KUKA KRL program: MyProgram_331().src

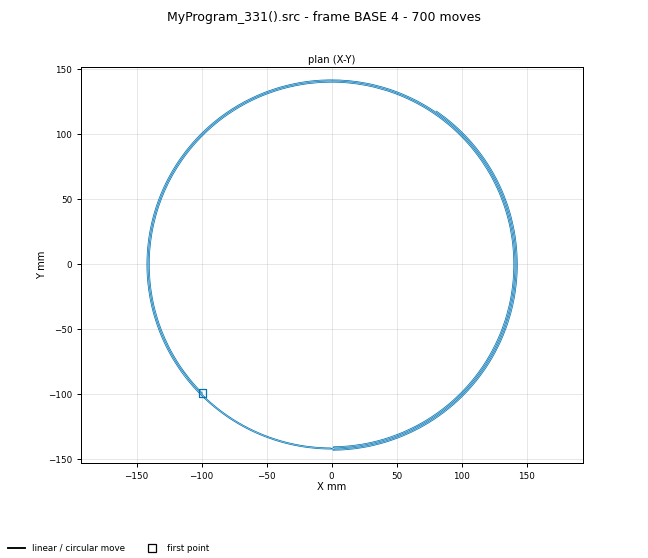
[picture p0: tool path of MyProgram_331().src in frame BASE 4, 700 of 700 moves have a stored position in this frame; points joined in program order, loops and branches not executed]
&ACCESS RVP
&REL 1
&PARAM TEMPLATE = C:\KRC\Roboter\Template\vorgabe
&PARAM EDITMASK = *
DEF MyProgram_331()
; ---- Setting reference (Base) ----
$BASE = BASE_DATA[4]

; --------------------------
; ---- Setting tool (TCP) ----
$TOOL = TOOL_DATA[3]
; --------------------------

$VEL.CP = VEL_APROX_PRINT
Startdeposition()
$VEL.CP = VEL_PRINT
LIN {X -99.2098,Y -99.0749,Z 188,A -128.7524,B 2.1644,C 0.244,E1 2.0676,E2 222.0446} C_DIS
LIN {X -102.5229,Y -95.6418,Z 188,A -131.099,B 2.1647,C 0.2414,E1 2.0629,E2 224.4451} C_DIS
LIN {X -106.6822,Y -90.9794,Z 188,A -133.6098,B 2.1653,C 0.2362,E1 2.0583,E2 226.9498} C_DIS
LIN {X -109.1006,Y -88.0645,Z 188,A -136.4618,B 2.1653,C 0.2366,E1 2.053,E2 229.9773} C_DIS
LIN {X -113.8783,Y -81.7931,Z 188,A -138.6384,B 2.1663,C 0.2268,E1 2.0496,E2 232.0127} C_DIS
LIN {X -116.0061,Y -78.7458,Z 188,A -140.3809,B 2.1666,C 0.224,E1 2.0468,E2 233.7852} C_DIS
LIN {X -118.4766,Y -74.9774,Z 188,A -142.4245,B 2.167,C 0.2203,E1 2.0437,E2 235.8555} C_DIS
LIN {X -121.0762,Y -70.7034,Z 188,A -144.5197,B 2.1674,C 0.2157,E1 2.0407,E2 237.9569} C_DIS
LIN {X -123.3353,Y -66.6846,Z 188,A -146.5209,B 2.1678,C 0.2114,E1 2.0379,E2 239.9733} C_DIS
LIN {X -125.1275,Y -63.2533,Z 188,A -148.0771,B 2.1682,C 0.2075,E1 2.036,E2 241.5254} C_DIS
LIN {X -126.6886,Y -60.0657,Z 188,A -149.6056,B 2.1685,C 0.2041,E1 2.0341,E2 243.0639} C_DIS
LIN {X -128.024,Y -57.1629,Z 188,A -151.3173,B 2.1688,C 0.2017,E1 2.0321,E2 244.8292} C_DIS
LIN {X -129.3709,Y -54.0455,Z 188,A -152.1682,B 2.1692,C 0.197,E1 2.0312,E2 245.6079} C_DIS
LIN {X -130.6105,Y -50.9774,Z 188,A -154.4978,B 2.1693,C 0.1957,E1 2.0287,E2 248.0671} C_DIS
LIN {X -132.2881,Y -46.4535,Z 188,A -155.8911,B 2.1699,C 0.1893,E1 2.0275,E2 249.3829} C_DIS
LIN {X -133.6605,Y -42.3408,Z 188,A -157.9257,B 2.1702,C 0.1852,E1 2.0257,E2 251.4516} C_DIS
LIN {X -134.6483,Y -39.0861,Z 188,A -159.3479,B 2.1705,C 0.1816,E1 2.0245,E2 252.8775} C_DIS
LIN {X -135.5192,Y -35.9493,Z 188,A -160.794,B 2.1708,C 0.1782,E1 2.0234,E2 254.3382} C_DIS
LIN {X -136.3712,Y -32.5697,Z 188,A -162.3237,B 2.1711,C 0.1746,E1 2.0224,E2 255.8812} C_DIS
LIN {X -137.2746,Y -28.5275,Z 188,A -164.3373,B 2.1714,C 0.1706,E1 2.0212,E2 257.9363} C_DIS
LIN {X -138.006,Y -24.7422,Z 188,A -165.7936,B 2.1718,C 0.166,E1 2.0205,E2 259.376} C_DIS
LIN {X -138.9297,Y -18.8902,Z 188,A -168.3319,B 2.1723,C 0.1595,E1 2.0194,E2 261.9286} C_DIS
LIN {X -139.6258,Y -12.7635,Z 188,A -171.0785,B 2.1727,C 0.1529,E1 2.0186,E2 264.7035} C_DIS
LIN {X -140.1378,Y -4.4233,Z 188,A -174.7771,B 2.1734,C 0.1439,E1 2.018,E2 268.4372} C_DIS
LIN {X -140.1787,Y 2.8448,Z 188,A -177.7366,B 2.1739,C 0.1356,E1 2.018,E2 271.3936} C_DIS
LIN {X -140.0302,Y 7.0299,Z 188,A -179.9971,B 2.1741,C 0.1317,E1 2.0182,E2 273.7241} C_DIS
LIN {X -139.782,Y 10.9262,Z 188,A 177.5471,B 2.1743,C 0.1288,E1 2.0189,E2 276.289} C_DIS
LIN {X -139.0996,Y 17.5935,Z 188,A 175.6823,B 2.1748,C 0.1196,E1 2.0194,E2 278.0404} C_DIS
LIN {X -138.1989,Y 23.6481,Z 188,A 172.9731,B 2.1752,C 0.1131,E1 2.0206,E2 280.7748} C_DIS
LIN {X -137.7195,Y 26.2897,Z 188,A 171.6814,B 2.1753,C 0.1104,E1 2.0212,E2 282.0906} C_DIS
LIN {X -136.8646,Y 30.4385,Z 188,A 169.7202,B 2.1755,C 0.106,E1 2.0224,E2 284.0801} C_DIS
LIN {X -135.2027,Y 37.1276,Z 188,A 166.9626,B 2.1759,C 0.0983,E1 2.0243,E2 286.8282} C_DIS
LIN {X -133.9173,Y 41.5233,Z 188,A 164.9103,B 2.1761,C 0.0936,E1 2.0259,E2 288.9021} C_DIS
LIN {X -132.743,Y 45.1415,Z 188,A 162.9991,B 2.1763,C 0.0902,E1 2.0277,E2 290.8574} C_DIS
LIN {X -131.3372,Y 49.0744,Z 188,A 161.3898,B 2.1764,C 0.0855,E1 2.0292,E2 292.4532} C_DIS
LIN {X -129.9982,Y 52.5188,Z 188,A 159.1417,B 2.1765,C 0.083,E1 2.0317,E2 294.7928} C_DIS
LIN {X -127.9992,Y 57.2184,Z 188,A 157.617,B 2.1768,C 0.0766,E1 2.0333,E2 296.2456} C_DIS
LIN {X -125.6046,Y 62.3001,Z 188,A 155.1346,B 2.177,C 0.0712,E1 2.0363,E2 298.7499} C_DIS
LIN {X -123.9945,Y 65.4459,Z 188,A 153.591,B 2.177,C 0.0679,E1 2.0383,E2 300.3049} C_DIS
LIN {X -121.9107,Y 69.2542,Z 188,A 150.9394,B 2.1771,C 0.0654,E1 2.0421,E2 303.0643} C_DIS
LIN {X -118.9504,Y 74.2235,Z 188,A 149.5886,B 2.1774,C 0.0578,E1 2.0439,E2 304.2876} C_DIS
LIN {X -114.8375,Y 80.4415,Z 188,A 145.4813,B 2.1774,C 0.0532,E1 2.0505,E2 308.5245} C_DIS
LIN {X -112.2475,Y 84.0171,Z 188,A 143.9413,B 2.1776,C 0.0486,E1 2.053,E2 310.0306} C_DIS
LIN {X -109.3338,Y 87.7754,Z 188,A 141.9211,B 2.1776,C 0.0446,E1 2.0565,E2 312.0589} C_DIS
LIN {X -106.409,Y 91.2989,Z 188,A 139.9971,B 2.1777,C 0.0409,E1 2.06,E2 313.9881} C_DIS
LIN {X -103.4782,Y 94.6081,Z 188,A 138.0511,B 2.1777,C 0.0376,E1 2.0636,E2 315.95} C_DIS
LIN {X -100.2471,Y 98.0248,Z 188,A 136.0546,B 2.1779,C 0.0341,E1 2.0675,E2 317.9543} C_DIS
LIN {X -96.8927,Y 101.3415,Z 188,A 134.0732,B 2.1779,C 0.0307,E1 2.0715,E2 319.9409} C_DIS
LIN {X -93.6314,Y 104.3622,Z 188,A 132.1553,B 2.1779,C 0.0277,E1 2.0755,E2 321.87} C_DIS
LIN {X -90.065,Y 107.455,Z 188,A 130.1679,B 2.1779,C 0.0245,E1 2.0797,E2 323.8631} C_DIS
LIN {X -86.4591,Y 110.3773,Z 188,A 128.1907,B 2.178,C 0.0217,E1 2.0841,E2 325.8488} C_DIS
LIN {X -82.9387,Y 113.0463,Z 188,A 126.1798,B 2.178,C 0.0195,E1 2.0886,E2 327.8835} C_DIS
LIN {X -78.3392,Y 116.2814,Z 188,A 124.065,B 2.178,C 0.0155,E1 2.0934,E2 329.9745} C_DIS
LIN {X -75.1994,Y 118.3365,Z 188,A 122.1429,B 2.178,C 0.0146,E1 2.0981,E2 331.9429} C_DIS
LIN {X -72.4256,Y 120.0535,Z 188,A 121.0215,B 2.178,C 0.0122,E1 2.1007,E2 333.0377} C_DIS
LIN {X -67.9868,Y 122.6217,Z 188,A 118.9997,B 2.178,C 0.0093,E1 2.1056,E2 335.0491} C_DIS
LIN {X -65.0011,Y 124.2281,Z 188,A 117.4444,B 2.1781,C 0.0083,E1 2.1095,E2 336.6242} C_DIS
LIN {X -60.611,Y 126.4281,Z 188,A 115.4931,B 2.1781,C 0.0059,E1 2.1144,E2 338.5675} C_DIS
LIN {X -56.8006,Y 128.1861,Z 188,A 113.2517,B 2.1781,C 0.0061,E1 2.1202,E2 340.8715} C_DIS
LIN {X -53.0986,Y 129.7645,Z 188,A 112.0341,B 2.1781,C 0.003,E1 2.1233,E2 342.0366} C_DIS
LIN {X -48.8586,Y 131.4181,Z 188,A 110.1163,B 2.1781,C 0.0017,E1 2.1283,E2 343.9603} C_DIS
LIN {X -45.7356,Y 132.537,Z 188,A 108.6718,B 2.1781,C 0.001,E1 2.1321,E2 345.4148} C_DIS
LIN {X -42.4483,Y 133.6262,Z 188,A 107.2892,B 2.1781,C -0.0001,E1 2.1358,E2 346.7926} C_DIS
LIN {X -39.4257,Y 134.5489,Z 188,A 105.9514,B 2.1781,C -0.0007,E1 2.1394,E2 348.1353} C_DIS
LIN {X -35.7551,Y 135.571,Z 188,A 104.4244,B 2.1781,C -0.0017,E1 2.1435,E2 349.6579} C_DIS
LIN {X -32.4671,Y 136.3959,Z 188,A 102.8487,B 2.1781,C -0.0017,E1 2.1478,E2 351.2558} C_DIS
LIN {X -27.1987,Y 137.545,Z 188,A 100.6704,B 2.1781,C -0.0026,E1 2.1538,E2 353.4301} C_DIS
LIN {X -21.4182,Y 138.5608,Z 188,A 98.2309,B 2.1781,C -0.0031,E1 2.1606,E2 355.8732} C_DIS
LIN {X -16.8516,Y 139.1903,Z 188,A 96.4114,B 2.1781,C -0.0037,E1 2.1656,E2 357.684} C_DIS
LIN {X -13.2817,Y 139.576,Z 188,A 95.0228,B 2.1781,C -0.0042,E1 2.1694,E2 359.0625} C_DIS
LIN {X -10.1301,Y 139.8401,Z 188,A 93.6605,B 2.1781,C -0.0039,E1 2.1732,E2 360.4326} C_DIS
LIN {X -5.9088,Y 140.0827,Z 188,A 91.9352,B 2.1781,C -0.0039,E1 2.1781,E2 362.1568} C_DIS
LIN {X -2.3359,Y 140.1871,Z 188,A 90.4902,B 2.1781,C -0.0038,E1 2.1821,E2 363.5993} C_DIS
LIN {X 1.1147,Y 140.2026,Z 188,A 89.0223,B 2.1781,C -0.0032,E1 2.1862,E2 365.0736} C_DIS
LIN {X 5.5113,Y 140.0982,Z 188,A 87.3185,B 2.1781,C -0.0032,E1 2.191,E2 366.7654} C_DIS
LIN {X 9.2429,Y 139.9029,Z 188,A 85.6697,B 2.1781,C -0.002,E1 2.1956,E2 368.4285} C_DIS
LIN {X 13.2851,Y 139.5757,Z 188,A 84.1627,B 2.1781,C -0.002,E1 2.1998,E2 369.9166} C_DIS
LIN {X 16.791,Y 139.1975,Z 188,A 82.7463,B 2.1781,C -0.0015,E1 2.2037,E2 371.3295} C_DIS
LIN {X 20.0562,Y 138.7647,Z 188,A 81.4071,B 2.1781,C -0.0007,E1 2.2074,E2 372.6675} C_DIS
LIN {X 23.8465,Y 138.1658,Z 188,A 79.8604,B 2.1781,C 0.0002,E1 2.2117,E2 374.2112} C_DIS
LIN {X 26.906,Y 137.6017,Z 188,A 78.305,B 2.1781,C 0.0026,E1 2.216,E2 375.8005} C_DIS
LIN {X 30.1812,Y 136.9196,Z 188,A 77.293,B 2.1781,C 0.0017,E1 2.2187,E2 376.7691} C_DIS
LIN {X 32.9842,Y 136.2712,Z 188,A 76.0874,B 2.1781,C 0.0028,E1 2.222,E2 377.978} C_DIS
LIN {X 42.4149,Y 133.6369,Z 188,A 72.4099,B 2.1781,C 0.0048,E1 2.2318,E2 381.6152} C_DIS
LIN {X 46.0947,Y 132.4125,Z 188,A 70.631,B 2.1781,C 0.0076,E1 2.2366,E2 383.4175} C_DIS
LIN {X 49.4775,Y 131.1862,Z 188,A 69.2128,B 2.1781,C 0.0089,E1 2.2403,E2 384.8291} C_DIS
LIN {X 52.7522,Y 129.9041,Z 188,A 67.8363,B 2.1781,C 0.0103,E1 2.2438,E2 386.1979} C_DIS
LIN {X 55.965,Y 128.5526,Z 188,A 66.4212,B 2.1781,C 0.012,E1 2.2475,E2 387.6117} C_DIS
LIN {X 59.0901,Y 127.1462,Z 188,A 65.0645,B 2.1781,C 0.0136,E1 2.2509,E2 388.9628} C_DIS
LIN {X 62.7,Y 125.4073,Z 188,A 63.4838,B 2.1781,C 0.0155,E1 2.2549,E2 390.5365} C_DIS
LIN {X 66.4011,Y 123.4876,Z 188,A 61.7566,B 2.1781,C 0.0182,E1 2.2591,E2 392.2664} C_DIS
LIN {X 70.4561,Y 121.22,Z 188,A 59.9224,B 2.1781,C 0.0206,E1 2.2636,E2 394.0926} C_DIS
LIN {X 74.3344,Y 118.8814,Z 188,A 58.1619,B 2.178,C 0.023,E1 2.2677,E2 395.8419} C_DIS
LIN {X 78.5545,Y 116.1356,Z 188,A 55.7652,B 2.178,C 0.0287,E1 2.2734,E2 398.2801} C_DIS
LIN {X 82.2259,Y 113.5658,Z 188,A 54.5625,B 2.178,C 0.0278,E1 2.276,E2 399.4055} C_DIS
LIN {X 85.2382,Y 111.3227,Z 188,A 52.9427,B 2.1779,C 0.0311,E1 2.2796,E2 401.0359} C_DIS
LIN {X 88.7755,Y 108.5228,Z 188,A 51.1831,B 2.1779,C 0.034,E1 2.2834,E2 402.7852} C_DIS
LIN {X 92.1501,Y 105.6723,Z 188,A 49.1657,B 2.1778,C 0.0389,E1 2.2878,E2 404.8289} C_DIS
LIN {X 94.9423,Y 103.1707,Z 188,A 48.0033,B 2.1778,C 0.0394,E1 2.2901,E2 405.9457} C_DIS
LIN {X 98.0757,Y 100.1972,Z 188,A 46.268,B 2.1777,C 0.0428,E1 2.2936,E2 407.6775} C_DIS
LIN {X 101.3708,Y 96.862,Z 188,A 44.4572,B 2.1777,C 0.0461,E1 2.2971,E2 409.4754} C_DIS
LIN {X 104.5155,Y 93.4602,Z 188,A 42.6598,B 2.1776,C 0.0495,E1 2.3004,E2 411.2612} C_DIS
LIN {X 107.5194,Y 89.9883,Z 188,A 40.5839,B 2.1774,C 0.0551,E1 2.3042,E2 413.3623} C_DIS
LIN {X 109.9426,Y 87.0102,Z 188,A 39.3934,B 2.1774,C 0.0559,E1 2.3062,E2 414.5059} C_DIS
LIN {X 112.7226,Y 83.3793,Z 188,A 37.5719,B 2.1773,C 0.0598,E1 2.3093,E2 416.3219} C_DIS
LIN {X 115.7769,Y 79.0829,Z 188,A 35.1908,B 2.1771,C 0.0666,E1 2.3131,E2 418.7319} C_DIS
LIN {X 118.1906,Y 75.4275,Z 188,A 34.1102,B 2.1771,C 0.0656,E1 2.3146,E2 419.7238} C_DIS
LIN {X 119.7881,Y 72.8644,Z 188,A 32.6774,B 2.177,C 0.0701,E1 2.3167,E2 421.182} C_DIS
LIN {X 122.0603,Y 68.9905,Z 188,A 30.9227,B 2.1769,C 0.0741,E1 2.3192,E2 422.9271} C_DIS
LIN {X 124.1823,Y 65.0882,Z 188,A 29.293,B 2.1768,C 0.0772,E1 2.3213,E2 424.5339} C_DIS
LIN {X 126.0478,Y 61.4016,Z 188,A 27.752,B 2.1766,C 0.0804,E1 2.3232,E2 426.0568} C_DIS
LIN {X 127.3901,Y 58.5626,Z 188,A 26.5205,B 2.1766,C 0.0833,E1 2.3246,E2 427.2821} C_DIS
LIN {X 128.8841,Y 55.1984,Z 188,A 25.1087,B 2.1764,C 0.0865,E1 2.3262,E2 428.6826} C_DIS
LIN {X 130.1851,Y 52.0551,Z 188,A 23.7748,B 2.1763,C 0.0897,E1 2.3276,E2 430.0098} C_DIS
LIN {X 131.5144,Y 48.6015,Z 188,A 22.4039,B 2.1762,C 0.0926,E1 2.3289,E2 431.3634} C_DIS
LIN {X 132.4961,Y 45.8535,Z 188,A 21.261,B 2.176,C 0.0954,E1 2.33,E2 432.5004} C_DIS
LIN {X 133.5958,Y 42.5433,Z 188,A 19.9102,B 2.1759,C 0.0986,E1 2.3312,E2 433.8422} C_DIS
LIN {X 134.6128,Y 39.2071,Z 188,A 18.1529,B 2.1756,C 0.1051,E1 2.3326,E2 435.6427} C_DIS
LIN {X 135.7427,Y 35.1014,Z 188,A 17.0085,B 2.1756,C 0.1051,E1 2.3333,E2 436.7114} C_DIS
LIN {X 136.7633,Y 30.8825,Z 188,A 14.9734,B 2.1752,C 0.1121,E1 2.3346,E2 438.7811} C_DIS
LIN {X 137.4849,Y 27.4941,Z 188,A 14.0857,B 2.1752,C 0.1118,E1 2.3351,E2 439.6013} C_DIS
LIN {X 138.1915,Y 23.6893,Z 188,A 12.4059,B 2.175,C 0.1169,E1 2.336,E2 441.2948} C_DIS
LIN {X 138.6247,Y 21.0053,Z 188,A 11.4004,B 2.1749,C 0.1192,E1 2.3364,E2 442.2872} C_DIS
LIN {X 139.1828,Y 16.9138,Z 188,A 9.8111,B 2.1746,C 0.1231,E1 2.3369,E2 443.8646} C_DIS
LIN {X 139.57,Y 13.3444,Z 188,A 8.4194,B 2.1744,C 0.1266,E1 2.3373,E2 445.2472} C_DIS
LIN {X 139.859,Y 9.8716,Z 188,A 7.127,B 2.1743,C 0.1295,E1 2.3376,E2 446.5233} C_DIS
LIN {X 140.0358,Y 6.9178,Z 188,A 5.927,B 2.1741,C 0.1328,E1 2.3378,E2 447.7228} C_DIS
LIN {X 140.1837,Y 2.5457,Z 188,A 4.2522,B 2.1738,C 0.1369,E1 2.3379,E2 449.3839} C_DIS
LIN {X 140.1955,Y -1.8311,Z 188,A 2.5476,B 2.1735,C 0.1413,E1 2.3379,E2 451.0786} C_DIS
LIN {X 140.078,Y -6.0282,Z 188,A 1.0433,B 2.1733,C 0.1444,E1 2.3378,E2 452.5562} C_DIS
LIN {X 139.9172,Y -9.0111,Z 188,A -0.2064,B 2.1731,C 0.148,E1 2.3376,E2 453.8105} C_DIS
LIN {X 139.5757,Y -13.2851,Z 188,A -1.7918,B 2.1728,C 0.1516,E1 2.3372,E2 455.375} C_DIS
LIN {X 139.1931,Y -16.8274,Z 188,A -3.1723,B 2.1726,C 0.155,E1 2.3367,E2 456.7464} C_DIS
LIN {X 138.6419,Y -20.8942,Z 188,A -4.8381,B 2.1723,C 0.1596,E1 2.3361,E2 458.4119} C_DIS
LIN {X 138.0023,Y -24.7629,Z 188,A -6.254,B 2.172,C 0.1625,E1 2.3354,E2 459.8042} C_DIS
LIN {X 137.3545,Y -28.1352,Z 188,A -7.6156,B 2.1718,C 0.1661,E1 2.3347,E2 461.1612} C_DIS
LIN {X 136.5408,Y -31.8563,Z 188,A -9.558,B 2.1712,C 0.1735,E1 2.3334,E2 463.1559} C_DIS
LIN {X 135.366,Y -36.5241,Z 188,A -10.524,B 2.1714,C 0.1708,E1 2.3329,E2 463.9901} C_DIS
LIN {X 134.6178,Y -39.1903,Z 188,A -11.9644,B 2.171,C 0.1763,E1 2.3317,E2 465.4727} C_DIS
LIN {X 133.5755,Y -42.6071,Z 188,A -13.7149,B 2.1705,C 0.1826,E1 2.3302,E2 467.263} C_DIS
LIN {X 132.2421,Y -46.5861,Z 188,A -14.909,B 2.1705,C 0.183,E1 2.3292,E2 468.3889} C_DIS
LIN {X 131.1909,Y -49.4649,Z 188,A -16.1267,B 2.1702,C 0.1861,E1 2.328,E2 469.6028} C_DIS
LIN {X 129.8527,Y -52.8798,Z 188,A -17.5174,B 2.1699,C 0.1892,E1 2.3266,E2 470.9802} C_DIS
LIN {X 128.5165,Y -56.0486,Z 188,A -18.8536,B 2.1696,C 0.1923,E1 2.3251,E2 472.3082} C_DIS
LIN {X 126.4213,Y -60.6253,Z 188,A -20.853,B 2.1692,C 0.1971,E1 2.3228,E2 474.3013} C_DIS
LIN {X 124.6261,Y -64.2382,Z 188,A -22.3339,B 2.1689,C 0.2,E1 2.3209,E2 475.761} C_DIS
LIN {X 123.1387,Y -67.0461,Z 188,A -23.7045,B 2.1686,C 0.2038,E1 2.3191,E2 477.1422} C_DIS
LIN {X 120.2001,Y -72.1824,Z 188,A -26.1333,B 2.168,C 0.2099,E1 2.3157,E2 479.5744} C_DIS
LIN {X 118.4571,Y -75.0083,Z 188,A -27.2434,B 2.1679,C 0.2113,E1 2.3141,E2 480.6522} C_DIS
LIN {X 115.8878,Y -78.9206,Z 188,A -29.0715,B 2.1675,C 0.2152,E1 2.3112,E2 482.4704} C_DIS
LIN {X 113.22,Y -82.7023,Z 188,A -30.8595,B 2.1671,C 0.2189,E1 2.3083,E2 484.2458} C_DIS
LIN {X 110.5284,Y -86.2668,Z 188,A -32.5985,B 2.1667,C 0.2224,E1 2.3054,E2 485.9745} C_DIS
LIN {X 107.6492,Y -89.8336,Z 188,A -34.3752,B 2.1664,C 0.2259,E1 2.3023,E2 487.7395} C_DIS
LIN {X 104.7094,Y -93.2437,Z 188,A -36.1267,B 2.166,C 0.2293,E1 2.2991,E2 489.4804} C_DIS
LIN {X 101.6866,Y -96.5314,Z 188,A -37.8777,B 2.1657,C 0.2326,E1 2.2957,E2 491.2227} C_DIS
LIN {X 98.4415,Y -99.8384,Z 188,A -39.6728,B 2.1653,C 0.2358,E1 2.2922,E2 493.0058} C_DIS
LIN {X 95.1717,Y -102.9602,Z 188,A -41.4428,B 2.165,C 0.239,E1 2.2886,E2 494.7666} C_DIS
LIN {X 91.7922,Y -105.9841,Z 188,A -43.2072,B 2.1646,C 0.242,E1 2.2849,E2 496.5204} C_DIS
LIN {X 88.2964,Y -108.9136,Z 188,A -45.0055,B 2.1643,C 0.2451,E1 2.2811,E2 498.3111} C_DIS
LIN {X 84.6418,Y -111.7771,Z 188,A -46.7989,B 2.164,C 0.2478,E1 2.2771,E2 500.0917} C_DIS
LIN {X 80.9701,Y -114.4647,Z 188,A -48.5935,B 2.1637,C 0.2507,E1 2.2731,E2 501.8788} C_DIS
LIN {X 77.1381,Y -117.0812,Z 188,A -50.3998,B 2.1633,C 0.2533,E1 2.2689,E2 503.674} C_DIS
LIN {X 73.415,Y -119.451,Z 188,A -52.1408,B 2.1631,C 0.2558,E1 2.2648,E2 505.4078} C_DIS
LIN {X 69.5513,Y -121.7412,Z 188,A -54.3796,B 2.1624,C 0.2615,E1 2.2592,E2 507.7034} C_DIS
LIN {X 65.297,Y -124.0727,Z 188,A -55.4851,B 2.1627,C 0.2584,E1 2.2568,E2 508.6893} C_DIS
LIN {X 62.3456,Y -125.5821,Z 188,A -57.9697,B 2.1616,C 0.268,E1 2.2502,E2 511.3306} C_DIS
LIN {X 55.9523,Y -128.5581,Z 188,A -59.6588,B 2.1621,C 0.2638,E1 2.2463,E2 512.8574} C_DIS
LIN {X 51.8433,Y -130.2705,Z 188,A -61.5908,B 2.1617,C 0.2669,E1 2.2412,E2 514.8064} C_DIS
LIN {X 48.8684,Y -131.4144,Z 188,A -62.8656,B 2.1615,C 0.2682,E1 2.2379,E2 516.0783} C_DIS
LIN {X 45.6831,Y -132.5552,Z 188,A -64.2683,B 2.1613,C 0.2699,E1 2.2342,E2 517.4847} C_DIS
LIN {X 40.0329,Y -134.3711,Z 188,A -66.523,B 2.1612,C 0.2713,E1 2.2282,E2 519.7173} C_DIS
LIN {X 35.6997,Y -135.5858,Z 188,A -68.3924,B 2.1609,C 0.2732,E1 2.2232,E2 521.592} C_DIS
LIN {X 31.5277,Y -136.6159,Z 188,A -70.398,B 2.1605,C 0.2763,E1 2.2176,E2 523.6333} C_DIS
LIN {X 28.2637,Y -137.3283,Z 188,A -71.6744,B 2.1605,C 0.2768,E1 2.2141,E2 524.8982} C_DIS
LIN {X 23.2299,Y -138.2687,Z 188,A -73.5037,B 2.1605,C 0.2767,E1 2.2092,E2 526.6921} C_DIS
LIN {X 19.8997,Y -138.787,Z 188,A -74.8474,B 2.1604,C 0.2774,E1 2.2055,E2 528.032} C_DIS
LIN {X 16.647,Y -139.2147,Z 188,A -76.1595,B 2.1604,C 0.278,E1 2.2019,E2 529.3409} C_DIS
LIN {X 13.5211,Y -139.553,Z 188,A -77.5172,B 2.1602,C 0.279,E1 2.198,E2 530.7095} C_DIS
LIN {X 9.6236,Y -139.8771,Z 188,A -79.1678,B 2.1601,C 0.28,E1 2.1934,E2 532.3683} C_DIS
LIN {X 5.5247,Y -140.0977,Z 188,A -80.7201,B 2.1601,C 0.2799,E1 2.1891,E2 533.9039} C_DIS
LIN {X 1.604,Y -140.1993,Z 188,A -82.3886,B 2.16,C 0.2807,E1 2.1844,E2 535.5824} C_DIS
LIN {X 1.604,Y -140.1993,Z 188,A -82.3886,B 2.16,C 0.2807,E1 2.1844,E2 535.5824} C_DIS
Enddeposition()
LIN {X 1.0301,Y -141.1013,Z 188,A -82.2979,B 2.0515,C 0.2751,E1 2.076,E2 535.5067} C_DIS
Startdeposition()
$VEL.CP = VEL_PRINT
LIN {X 5.1326,Y -141.013,Z 188,A -79.9861,B 2.052,C 0.2712,E1 2.0828,E2 533.1027} C_DIS
LIN {X 8.9175,Y -140.824,Z 188,A -78.4272,B 2.052,C 0.2705,E1 2.0871,E2 531.5401} C_DIS
LIN {X 13.2109,Y -140.4863,Z 188,A -76.7454,B 2.0521,C 0.27,E1 2.0918,E2 529.8669} C_DIS
LIN {X 16.6843,Y -140.1159,Z 188,A -75.3233,B 2.0522,C 0.2692,E1 2.0958,E2 528.4434} C_DIS
LIN {X 21.0632,Y -139.5258,Z 188,A -73.5342,B 2.0524,C 0.2681,E1 2.1007,E2 526.6541} C_DIS
LIN {X 25.5651,Y -138.7723,Z 188,A -71.0714,B 2.053,C 0.2632,E1 2.1078,E2 524.1032} C_DIS
LIN {X 31.1897,Y -137.6156,Z 188,A -69.7147,B 2.0525,C 0.2672,E1 2.1111,E2 522.884} C_DIS
LIN {X 34.39,Y -136.8511,Z 188,A -67.9711,B 2.053,C 0.2635,E1 2.116,E2 521.0818} C_DIS
LIN {X 38.6394,Y -135.7137,Z 188,A -66.4394,B 2.053,C 0.2634,E1 2.12,E2 519.5851} C_DIS
LIN {X 44.0088,Y -134.0684,Z 188,A -64.1787,B 2.0533,C 0.2611,E1 2.1261,E2 517.3258} C_DIS
LIN {X 47.4967,Y -132.8719,Z 188,A -62.7488,B 2.0534,C 0.2599,E1 2.1298,E2 515.9044} C_DIS
LIN {X 50.7185,Y -131.676,Z 188,A -61.3884,B 2.0536,C 0.2584,E1 2.1334,E2 514.548} C_DIS
LIN {X 54.1566,Y -130.2991,Z 188,A -60.0104,B 2.0538,C 0.2574,E1 2.1369,E2 513.1868} C_DIS
LIN {X 57.2498,Y -128.9703,Z 188,A -57.972,B 2.0545,C 0.2512,E1 2.1424,E2 511.0521} C_DIS
LIN {X 62.2293,Y -126.6423,Z 188,A -56.4621,B 2.0543,C 0.2528,E1 2.1459,E2 509.6432} C_DIS
LIN {X 68.9463,Y -123.1168,Z 188,A -53.3804,B 2.0549,C 0.2482,E1 2.1535,E2 506.5593} C_DIS
LIN {X 72.9077,Y -120.813,Z 188,A -51.606,B 2.0552,C 0.2459,E1 2.1577,E2 504.7957} C_DIS
LIN {X 76.8278,Y -118.3587,Z 188,A -49.8126,B 2.0555,C 0.2433,E1 2.162,E2 503.0128} C_DIS
LIN {X 80.7439,Y -115.7227,Z 188,A -47.9749,B 2.0558,C 0.2405,E1 2.1662,E2 501.1848} C_DIS
LIN {X 84.5098,Y -113.0021,Z 188,A -46.1617,B 2.0561,C 0.2377,E1 2.1702,E2 499.3805} C_DIS
LIN {X 88.1524,Y -110.1842,Z 188,A -44.3662,B 2.0565,C 0.2347,E1 2.1742,E2 497.5941} C_DIS
LIN {X 91.6613,Y -107.2828,Z 188,A -42.5914,B 2.0568,C 0.2317,E1 2.1779,E2 495.8282} C_DIS
LIN {X 95.1386,Y -104.2119,Z 188,A -40.7879,B 2.0572,C 0.2285,E1 2.1817,E2 494.0345} C_DIS
LIN {X 98.4926,Y -101.0479,Z 188,A -38.9842,B 2.0575,C 0.2251,E1 2.1853,E2 492.239} C_DIS
LIN {X 101.7583,Y -97.7582,Z 188,A -37.2171,B 2.0579,C 0.222,E1 2.1887,E2 490.4865} C_DIS
LIN {X 104.8541,Y -94.4302,Z 188,A -35.4678,B 2.0582,C 0.2187,E1 2.192,E2 488.7493} C_DIS
LIN {X 107.7751,Y -91.0822,Z 188,A -33.7521,B 2.0586,C 0.2154,E1 2.1951,E2 487.0445} C_DIS
LIN {X 110.687,Y -87.5207,Z 188,A -31.966,B 2.059,C 0.2118,E1 2.1982,E2 485.2683} C_DIS
LIN {X 113.4761,Y -83.8727,Z 188,A -30.2057,B 2.0593,C 0.2082,E1 2.2011,E2 483.5211} C_DIS
LIN {X 116.1443,Y -80.1368,Z 188,A -28.4385,B 2.0597,C 0.2045,E1 2.204,E2 481.7659} C_DIS
LIN {X 118.7112,Y -76.2823,Z 188,A -26.8391,B 2.0599,C 0.2022,E1 2.2063,E2 480.2039} C_DIS
LIN {X 122.4713,Y -70.0865,Z 188,A -24.2243,B 2.0604,C 0.1975,E1 2.2101,E2 477.6323} C_DIS
LIN {X 124.0074,Y -67.3316,Z 188,A -22.5437,B 2.061,C 0.1911,E1 2.2124,E2 475.8956} C_DIS
LIN {X 126.2721,Y -62.9798,Z 188,A -20.3983,B 2.0615,C 0.1848,E1 2.2151,E2 473.7274} C_DIS
LIN {X 128.3745,Y -58.5766,Z 188,A -18.9446,B 2.0616,C 0.1839,E1 2.2167,E2 472.3451} C_DIS
LIN {X 130.085,Y -54.6691,Z 188,A -17.4086,B 2.0619,C 0.1809,E1 2.2184,E2 470.8347} C_DIS
LIN {X 131.4381,Y -51.3305,Z 188,A -16.151,B 2.0621,C 0.1786,E1 2.2197,E2 469.6041} C_DIS
LIN {X 132.6222,Y -48.1893,Z 188,A -14.7696,B 2.0624,C 0.1749,E1 2.221,E2 468.2192} C_DIS
LIN {X 133.9799,Y -44.2747,Z 188,A -12.8566,B 2.0629,C 0.1685,E1 2.2227,E2 466.2734} C_DIS
LIN {X 135.1383,Y -40.6069,Z 188,A -11.6072,B 2.0631,C 0.1668,E1 2.2237,E2 465.0657} C_DIS
LIN {X 136.0725,Y -37.3564,Z 188,A -10.1383,B 2.0634,C 0.1623,E1 2.2248,E2 463.5827} C_DIS
LIN {X 136.9755,Y -33.8988,Z 188,A -8.9708,B 2.0636,C 0.1606,E1 2.2256,E2 462.4529} C_DIS
LIN {X 137.8178,Y -30.2872,Z 188,A -7.7769,B 2.0637,C 0.1589,E1 2.2263,E2 461.3002} C_DIS
LIN {X 138.4986,Y -27.0039,Z 188,A -6.3312,B 2.064,C 0.1545,E1 2.2271,E2 459.8422} C_DIS
LIN {X 139.1503,Y -23.4102,Z 188,A -4.9791,B 2.0643,C 0.1514,E1 2.2277,E2 458.5068} C_DIS
LIN {X 139.8155,Y -19.0522,Z 188,A -3.2109,B 2.0646,C 0.1466,E1 2.2284,E2 456.7403} C_DIS
LIN {X 140.2828,Y -15.2177,Z 188,A -1.8268,B 2.0648,C 0.1437,E1 2.2289,E2 455.3801} C_DIS
LIN {X 140.6617,Y -11.2065,Z 188,A -0.2099,B 2.0651,C 0.1393,E1 2.2293,E2 453.7647} C_DIS
LIN {X 140.9231,Y -7.1804,Z 188,A 1.2213,B 2.0653,C 0.1363,E1 2.2295,E2 452.3602} C_DIS
LIN {X 141.062,Y -3.5416,Z 188,A 2.6596,B 2.0656,C 0.1325,E1 2.2296,E2 450.9264} C_DIS
LIN {X 141.1068,Y 0.4422,Z 188,A 4.1976,B 2.0658,C 0.1286,E1 2.2296,E2 449.3981} C_DIS
LIN {X 141.0427,Y 4.2343,Z 188,A 5.633,B 2.066,C 0.1251,E1 2.2296,E2 447.9758} C_DIS
LIN {X 140.8449,Y 8.5781,Z 188,A 7.22,B 2.0662,C 0.1216,E1 2.2293,E2 446.4116} C_DIS
LIN {X 140.5533,Y 12.4896,Z 188,A 8.8157,B 2.0665,C 0.1171,E1 2.2289,E2 444.8146} C_DIS
LIN {X 140.1726,Y 16.2095,Z 188,A 10.1871,B 2.0667,C 0.114,E1 2.2285,E2 443.4619} C_DIS
LIN {X 139.7427,Y 19.569,Z 188,A 11.3302,B 2.0667,C 0.112,E1 2.2281,E2 442.3488} C_DIS
LIN {X 139.2951,Y 22.5427,Z 188,A 12.786,B 2.0671,C 0.1068,E1 2.2274,E2 440.8613} C_DIS
LIN {X 138.417,Y 27.4238,Z 188,A 14.394,B 2.0671,C 0.1044,E1 2.2266,E2 439.306} C_DIS
LIN {X 136.8388,Y 34.4384,Z 188,A 17.8857,B 2.0678,C 0.0919,E1 2.2243,E2 435.7372} C_DIS
LIN {X 135.2451,Y 40.2481,Z 188,A 19.5701,B 2.0678,C 0.0913,E1 2.2231,E2 434.1524} C_DIS
LIN {X 134.0359,Y 44.1064,Z 188,A 21.056,B 2.0679,C 0.088,E1 2.2218,E2 432.6862} C_DIS
LIN {X 132.8543,Y 47.5455,Z 188,A 22.4337,B 2.0681,C 0.0849,E1 2.2206,E2 431.3208} C_DIS
LIN {X 131.7238,Y 50.5954,Z 188,A 23.6471,B 2.0681,C 0.0822,E1 2.2194,E2 430.1209} C_DIS
LIN {X 130.4366,Y 53.8273,Z 188,A 25.0417,B 2.0683,C 0.0786,E1 2.2179,E2 428.7281} C_DIS
LIN {X 128.9013,Y 57.4041,Z 188,A 26.4581,B 2.0684,C 0.0758,E1 2.2163,E2 427.3324} C_DIS
LIN {X 127.4367,Y 60.5861,Z 188,A 27.7932,B 2.0685,C 0.0728,E1 2.2148,E2 426.0081} C_DIS
LIN {X 125.9178,Y 63.6833,Z 188,A 29.1315,B 2.0686,C 0.0697,E1 2.2131,E2 424.6775} C_DIS
LIN {X 124.0999,Y 67.1617,Z 188,A 30.7324,B 2.0688,C 0.0656,E1 2.211,E2 423.0751} C_DIS
LIN {X 121.8302,Y 71.1954,Z 188,A 32.4882,B 2.0688,C 0.0618,E1 2.2086,E2 421.3347} C_DIS
LIN {X 119.5418,Y 74.9747,Z 188,A 34.0173,B 2.069,C 0.0594,E1 2.2064,E2 419.8393} C_DIS
LIN {X 116.7646,Y 79.2296,Z 188,A 36.0152,B 2.069,C 0.055,E1 2.2033,E2 417.8492} C_DIS
LIN {X 114.4115,Y 82.5915,Z 188,A 37.7202,B 2.0692,C 0.0508,E1 2.2006,E2 416.1389} C_DIS
LIN {X 112.1056,Y 85.6949,Z 188,A 39.4904,B 2.0693,C 0.0457,E1 2.1975,E2 414.3426} C_DIS
LIN {X 109.5461,Y 88.9446,Z 188,A 40.7717,B 2.0693,C 0.0448,E1 2.1954,E2 413.1122} C_DIS
LIN {X 106.683,Y 92.3588,Z 188,A 42.4543,B 2.0693,C 0.0417,E1 2.1923,E2 411.4454} C_DIS
LIN {X 103.8314,Y 95.5528,Z 188,A 44.1156,B 2.0695,C 0.0384,E1 2.1892,E2 409.7937} C_DIS
LIN {X 100.6907,Y 98.8568,Z 188,A 45.8758,B 2.0695,C 0.0352,E1 2.1858,E2 408.0448} C_DIS
LIN {X 97.4496,Y 102.0533,Z 188,A 47.4402,B 2.0695,C 0.0333,E1 2.1828,E2 406.5162} C_DIS
LIN {X 93.9524,Y 105.282,Z 188,A 49.499,B 2.0696,C 0.0286,E1 2.1785,E2 404.4413} C_DIS
LIN {X 90.5157,Y 108.2509,Z 188,A 51.2137,B 2.0696,C 0.0259,E1 2.1749,E2 402.7428} C_DIS
LIN {X 87.1753,Y 110.9583,Z 188,A 52.934,B 2.0696,C 0.0228,E1 2.1711,E2 401.0258} C_DIS
LIN {X 83.0199,Y 114.101,Z 188,A 55.1771,B 2.0697,C 0.0182,E1 2.166,E2 398.7665} C_DIS
LIN {X 80.1402,Y 116.142,Z 188,A 56.2344,B 2.0697,C 0.0182,E1 2.1637,E2 397.7566} C_DIS
LIN {X 76.6995,Y 118.442,Z 188,A 57.9421,B 2.0697,C 0.0152,E1 2.1597,E2 396.0456} C_DIS
LIN {X 72.7758,Y 120.8927,Z 188,A 59.7549,B 2.0697,C 0.0126,E1 2.1554,E2 394.241} C_DIS
LIN {X 68.7883,Y 123.2056,Z 188,A 61.5865,B 2.0697,C 0.0099,E1 2.151,E2 392.4147} C_DIS
LIN {X 64.445,Y 125.53,Z 188,A 63.4202,B 2.0697,C 0.008,E1 2.1465,E2 390.6019} C_DIS
LIN {X 61.1148,Y 127.1841,Z 188,A 64.8109,B 2.0698,C 0.0067,E1 2.143,E2 389.2263} C_DIS
LIN {X 58.0511,Y 128.6119,Z 188,A 66.2501,B 2.0698,C 0.0044,E1 2.1393,E2 387.7789} C_DIS
LIN {X 54.7479,Y 130.0521,Z 188,A 67.6665,B 2.0698,C 0.0029,E1 2.1357,E2 386.3686} C_DIS
LIN {X 51.4184,Y 131.4039,Z 188,A 69.0135,B 2.0698,C 0.0018,E1 2.1322,E2 385.0358} C_DIS
LIN {X 48.2435,Y 132.6027,Z 188,A 70.4026,B 2.0698,C 0.0001,E1 2.1286,E2 383.6455} C_DIS
LIN {X 44.7131,Y 133.8339,Z 188,A 71.8109,B 2.0698,C -0.0009,E1 2.1249,E2 382.2512} C_DIS
LIN {X 41.1512,Y 134.9717,Z 188,A 74.2305,B 2.0698,C -0.0075,E1 2.1181,E2 379.7193} C_DIS
LIN {X 34.5365,Y 136.8139,Z 188,A 76.0722,B 2.0698,C -0.0047,E1 2.1135,E2 377.9967} C_DIS
LIN {X 28.2349,Y 138.2519,Z 188,A 78.6075,B 2.0698,C -0.0063,E1 2.1066,E2 375.4732} C_DIS
LIN {X 23.6746,Y 139.1062,Z 188,A 80.5766,B 2.0698,C -0.0081,E1 2.1011,E2 373.4942} C_DIS
LIN {X 19.7324,Y 139.7194,Z 188,A 82.1304,B 2.0698,C -0.0087,E1 2.0968,E2 371.9491} C_DIS
LIN {X 15.4188,Y 140.2612,Z 188,A 83.8596,B 2.0698,C -0.0095,E1 2.092,E2 370.2249} C_DIS
LIN {X 11.7677,Y 140.6143,Z 188,A 85.3378,B 2.0698,C -0.0101,E1 2.0879,E2 368.7487} C_DIS
LIN {X 7.6714,Y 140.8984,Z 188,A 87.006,B 2.0698,C -0.0107,E1 2.0832,E2 367.081} C_DIS
LIN {X 4.0415,Y 141.0481,Z 188,A 88.416,B 2.0698,C -0.0109,E1 2.0793,E2 365.6795} C_DIS
LIN {X 0,Y 141.1081,Z 188,A 90.1398,B 2.0698,C -0.0116,E1 2.0745,E2 363.9463} C_DIS
LIN {X -3.8386,Y 141.0537,Z 188,A 91.649,B 2.0698,C -0.0116,E1 2.0703,E2 362.4438} C_DIS
LIN {X -8.3106,Y 140.8614,Z 188,A 93.3945,B 2.0698,C -0.0114,E1 2.0654,E2 360.708} C_DIS
LIN {X -11.755,Y 140.6154,Z 188,A 94.8663,B 2.0698,C -0.0117,E1 2.0613,E2 359.2283} C_DIS
LIN {X -15.9645,Y 140.2018,Z 188,A 96.6827,B 2.0698,C -0.0119,E1 2.0562,E2 357.4005} C_DIS
LIN {X -22.9441,Y 139.2281,Z 188,A 99.4307,B 2.0698,C -0.0108,E1 2.0486,E2 354.6679} C_DIS
LIN {X -26.4033,Y 138.6134,Z 188,A 100.793,B 2.0698,C -0.0101,E1 2.0449,E2 353.3142} C_DIS
LIN {X -30.8864,Y 137.6849,Z 188,A 102.7153,B 2.0698,C -0.0097,E1 2.0396,E2 351.3851} C_DIS
LIN {X -33.6347,Y 137.0395,Z 188,A 104.1123,B 2.0698,C -0.0101,E1 2.0357,E2 349.9578} C_DIS
LIN {X -37.8932,Y 135.9224,Z 188,A 105.7377,B 2.0698,C -0.0085,E1 2.0314,E2 348.3534} C_DIS
LIN {X -41.3336,Y 134.9159,Z 188,A 107.1591,B 2.0698,C -0.0075,E1 2.0276,E2 346.937} C_DIS
LIN {X -44.7199,Y 133.8316,Z 188,A 108.5247,B 2.0698,C -0.0062,E1 2.024,E2 345.5818} C_DIS
LIN {X -47.6096,Y 132.8312,Z 188,A 109.974,B 2.0698,C -0.006,E1 2.0201,E2 344.1077} C_DIS
LIN {X -51.089,Y 131.532,Z 188,A 111.4478,B 2.0698,C -0.0047,E1 2.0162,E2 342.639} C_DIS
LIN {X -57.2567,Y 128.9672,Z 188,A 114.1432,B 2.0698,C -0.0021,E1 2.0093,E2 339.9474} C_DIS
LIN {X -60.6808,Y 127.3915,Z 188,A 115.7116,B 2.0698,C -0.0007,E1 2.0053,E2 338.3752} C_DIS
LIN {X -64.7644,Y 125.3674,Z 188,A 117.8593,B 2.0698,C 0.0004,E1 1.9998,E2 336.1921} C_DIS
LIN {X -67.6232,Y 123.8483,Z 188,A 119.6938,B 2.0698,C 0.0004,E1 1.9952,E2 334.2937} C_DIS
LIN {X -72.1145,Y 121.2881,Z 188,A 121.2882,B 2.0698,C 0.0046,E1 1.9915,E2 332.7635} C_DIS
LIN {X -75.8175,Y 119.0088,Z 188,A 123.1492,B 2.0698,C 0.0066,E1 1.9871,E2 330.8919} C_DIS
LIN {X -79.6232,Y 116.4968,Z 188,A 125.3941,B 2.0698,C 0.0081,E1 1.9817,E2 328.5992} C_DIS
LIN {X -82.899,Y 114.1887,Z 188,A 126.7122,B 2.0698,C 0.0115,E1 1.9788,E2 327.3208} C_DIS
LIN {X -86.464,Y 111.5135,Z 188,A 128.6351,B 2.0698,C 0.014,E1 1.9745,E2 325.3851} C_DIS
LIN {X -90.1331,Y 108.5695,Z 188,A 130.6218,B 2.0698,C 0.017,E1 1.9702,E2 323.3901} C_DIS
LIN {X -93.7045,Y 105.5029,Z 188,A 132.5991,B 2.0698,C 0.0201,E1 1.966,E2 321.4058} C_DIS
LIN {X -97.0418,Y 102.4415,Z 188,A 134.4883,B 2.0697,C 0.0233,E1 1.9621,E2 319.5117} C_DIS
LIN {X -100.1289,Y 99.4257,Z 188,A 136.3491,B 2.0697,C 0.0263,E1 1.9584,E2 317.6384} C_DIS
LIN {X -103.0919,Y 96.3504,Z 188,A 138.2094,B 2.0697,C 0.0294,E1 1.9548,E2 315.7636} C_DIS
LIN {X -106.1361,Y 92.9865,Z 188,A 140.1596,B 2.0696,C 0.0328,E1 1.9512,E2 313.8011} C_DIS
LIN {X -109.0555,Y 89.5449,Z 188,A 142.1106,B 2.0695,C 0.0363,E1 1.9477,E2 311.8364} C_DIS
LIN {X -111.8888,Y 85.9784,Z 188,A 144.5247,B 2.0695,C 0.0391,E1 1.9434,E2 309.352} C_DIS
LIN {X -114.7573,Y 82.1099,Z 188,A 145.9909,B 2.0693,C 0.0444,E1 1.9411,E2 307.9494} C_DIS
LIN {X -117.6807,Y 77.863,Z 188,A 148.3487,B 2.0693,C 0.0486,E1 1.9374,E2 305.5596} C_DIS
LIN {X -120.1788,Y 73.9485,Z 188,A 150.9577,B 2.0692,C 0.0516,E1 1.9334,E2 302.8595} C_DIS
LIN {X -123.0081,Y 69.1397,Z 188,A 152.7035,B 2.069,C 0.058,E1 1.9311,E2 301.182} C_DIS
LIN {X -125.045,Y 65.3797,Z 188,A 154.5128,B 2.0689,C 0.0621,E1 1.9287,E2 299.3645} C_DIS
LIN {X -126.5299,Y 62.4572,Z 188,A 156.0706,B 2.0688,C 0.065,E1 1.9267,E2 297.7786} C_DIS
LIN {X -128.9459,Y 57.3043,Z 188,A 158.4412,B 2.0686,C 0.0707,E1 1.924,E2 295.402} C_DIS
LIN {X -130.8879,Y 52.717,Z 188,A 160.5291,B 2.0684,C 0.0758,E1 1.9217,E2 293.3072} C_DIS
LIN {X -132.1128,Y 49.5677,Z 188,A 161.9394,B 2.0683,C 0.0793,E1 1.9203,E2 291.893} C_DIS
LIN {X -133.1312,Y 46.7671,Z 188,A 163.5114,B 2.0682,C 0.0818,E1 1.9188,E2 290.2751} C_DIS
LIN {X -134.7809,Y 41.7746,Z 188,A 165.6014,B 2.068,C 0.0876,E1 1.917,E2 288.1925} C_DIS
LIN {X -135.7812,Y 38.3981,Z 188,A 166.9125,B 2.0678,C 0.0916,E1 1.916,E2 286.8977} C_DIS
LIN {X -136.5207,Y 35.6843,Z 188,A 168.7158,B 2.0677,C 0.0936,E1 1.9147,E2 285.0093} C_DIS
LIN {X -137.4263,Y 32.0185,Z 188,A 169.859,B 2.0675,C 0.0984,E1 1.914,E2 283.918} C_DIS
LIN {X -138.4087,Y 27.4644,Z 188,A 172.1256,B 2.0673,C 0.103,E1 1.9126,E2 281.6038} C_DIS
LIN {X -138.9668,Y 24.4785,Z 188,A 174.1602,B 2.0671,C 0.1051,E1 1.9117,E2 279.4646} C_DIS
LIN {X -139.8922,Y 18.4667,Z 188,A 175.6778,B 2.0667,C 0.1135,E1 1.9111,E2 278.0741} C_DIS
LIN {X -140.586,Y 12.103,Z 188,A 178.7918,B 2.0663,C 0.1199,E1 1.9102,E2 274.8944} C_DIS
LIN {X -141.0256,Y 4.7998,Z 188,A -177.8086,B 2.0659,C 0.1276,E1 1.9097,E2 271.4401} C_DIS
LIN {X -141.108,Y -0.2305,Z 188,A -175.7184,B 2.0655,C 0.1332,E1 1.9097,E2 269.345} C_DIS
LIN {X -141.0388,Y -4.3756,Z 188,A -174.1723,B 2.0652,C 0.1382,E1 1.9097,E2 267.818} C_DIS
LIN {X -140.7711,Y -9.7289,Z 188,A -171.5515,B 2.0648,C 0.1435,E1 1.9102,E2 265.1395} C_DIS
LIN {X -140.1726,Y -16.2087,Z 188,A -168.7925,B 2.0643,C 0.1507,E1 1.9109,E2 262.3664} C_DIS
LIN {X -139.5677,Y -20.7876,Z 188,A -166.389,B 2.064,C 0.155,E1 1.9119,E2 259.8929} C_DIS
LIN {X -138.9127,Y -24.7803,Z 188,A -165.2828,B 2.0636,C 0.1604,E1 1.9124,E2 258.8598} C_DIS
LIN {X -138.3996,Y -27.5094,Z 188,A -163.7699,B 2.0634,C 0.1628,E1 1.9132,E2 257.2958} C_DIS
LIN {X -137.5459,Y -31.4948,Z 188,A -162.107,B 2.063,C 0.1673,E1 1.9143,E2 255.6325} C_DIS
LIN {X -136.6532,Y -35.1697,Z 188,A -160.4494,B 2.0627,C 0.1713,E1 1.9154,E2 253.9593} C_DIS
LIN {X -135.5155,Y -39.3247,Z 188,A -158.5852,B 2.0623,C 0.1757,E1 1.9168,E2 252.0803} C_DIS
LIN {X -134.4659,Y -42.7751,Z 188,A -157.0205,B 2.062,C 0.1794,E1 1.9181,E2 250.5027} C_DIS
LIN {X -133.266,Y -46.3785,Z 188,A -154.8721,B 2.0618,C 0.1823,E1 1.9202,E2 248.2724} C_DIS
LIN {X -131.742,Y -50.5486,Z 188,A -153.4143,B 2.0613,C 0.1876,E1 1.9216,E2 246.8625} C_DIS
LIN {X -130.337,Y -54.0659,Z 188,A -151.8154,B 2.0609,C 0.1914,E1 1.9232,E2 245.2559} C_DIS
LIN {X -128.4487,Y -58.4155,Z 188,A -149.5923,B 2.0605,C 0.1957,E1 1.9258,E2 242.9929} C_DIS
LIN {X -126.7053,Y -62.1017,Z 188,A -147.9849,B 2.0601,C 0.1998,E1 1.9277,E2 241.3927} C_DIS
LIN {X -125.2522,Y -64.9852,Z 188,A -146.4992,B 2.0599,C 0.2027,E1 1.9297,E2 239.8835} C_DIS
LIN {X -123.0472,Y -69.0701,Z 188,A -144.4964,B 2.0595,C 0.2069,E1 1.9324,E2 237.8651} C_DIS
LIN {X -120.6392,Y -73.195,Z 188,A -142.5787,B 2.059,C 0.2115,E1 1.9351,E2 235.951} C_DIS
LIN {X -118.4553,Y -76.6789,Z 188,A -140.6715,B 2.0586,C 0.2147,E1 1.938,E2 234.0115} C_DIS
LIN {X -116.0486,Y -80.2754,Z 188,A -138.7748,B 2.0583,C 0.2183,E1 1.9411,E2 232.096} C_DIS
LIN {X -109.4431,Y -89.0706,Z 188,A -134.1552,B 2.0573,C 0.2275,E1 1.9489,E2 227.4564} C_DIS
LIN {X -105.4566,Y -93.7569,Z 188,A -131.4642,B 2.0568,C 0.2319,E1 1.9539,E2 224.7391} C_DIS
LIN {X -102.893,Y -96.5632,Z 188,A -129.8096,B 2.0565,C 0.2346,E1 1.9571,E2 223.0691} C_DIS
LIN {X -99.6159,Y -99.9401,Z 188,A -127.1562,B 2.0563,C 0.236,E1 1.9625,E2 220.3118} C_DIS
LIN {X -95.3331,Y -104.0333,Z 188,A -125.3605,B 2.0556,C 0.2421,E1 1.966,E2 218.6021} C_DIS
LIN {X -92.7811,Y -106.3154,Z 188,A -123.7514,B 2.0554,C 0.2438,E1 1.9695,E2 216.9624} C_DIS
LIN {X -88.7935,Y -109.668,Z 188,A -121.6502,B 2.055,C 0.2472,E1 1.974,E2 214.8632} C_DIS
LIN {X -85.1258,Y -112.5385,Z 188,A -119.4771,B 2.0548,C 0.2492,E1 1.9789,E2 212.6505} C_DIS
LIN {X -82.3,Y -114.6214,Z 188,A -118.3937,B 2.0544,C 0.2525,E1 1.9813,E2 211.6152} C_DIS
LIN {X -79.3419,Y -116.6886,Z 188,A -116.6772,B 2.0542,C 0.2537,E1 1.9853,E2 209.8634} C_DIS
LIN {X -75.5594,Y -119.1728,Z 188,A -114.7873,B 2.0539,C 0.256,E1 1.9898,E2 207.9659} C_DIS
LIN {X -71.6938,Y -121.5374,Z 188,A -112.8915,B 2.0537,C 0.2581,E1 1.9943,E2 206.0621} C_DIS
LIN {X -67.6247,Y -123.8475,Z 188,A -111.0503,B 2.0534,C 0.2605,E1 1.9988,E2 204.229} C_DIS
LIN {X -64.4192,Y -125.5432,Z 188,A -109.512,B 2.0532,C 0.2619,E1 2.0027,E2 202.6811} C_DIS
LIN {X -61.1485,Y -127.168,Z 188,A -108.0132,B 2.053,C 0.2634,E1 2.0065,E2 201.1798} C_DIS
LIN {X -57.8698,Y -128.693,Z 188,A -106.5191,B 2.0528,C 0.2647,E1 2.0103,E2 199.6818} C_DIS
LIN {X -54.7279,Y -130.0605,Z 188,A -105.0564,B 2.0528,C 0.2656,E1 2.0141,E2 198.2088} C_DIS
LIN {X -51.6758,Y -131.3038,Z 188,A -103.7454,B 2.0525,C 0.2669,E1 2.0175,E2 196.9013} C_DIS
LIN {X -48.0876,Y -132.6589,Z 188,A -102.3187,B 2.0523,C 0.2686,E1 2.0212,E2 195.4927} C_DIS
LIN {X -44.4695,Y -133.915,Z 188,A -100.3652,B 2.0524,C 0.268,E1 2.0265,E2 193.4824} C_DIS
LIN {X -38.9645,Y -135.621,Z 188,A -98.0428,B 2.0522,C 0.2694,E1 2.0327,E2 191.162} C_DIS
LIN {X -35.3792,Y -136.6,Z 188,A -96.1412,B 2.0523,C 0.2684,E1 2.038,E2 189.204} C_DIS
LIN {X -30.9953,Y -137.66,Z 188,A -94.7271,B 2.052,C 0.271,E1 2.0417,E2 187.8487} C_DIS
LIN {X -26.7461,Y -138.5479,Z 188,A -93.0137,B 2.0519,C 0.2718,E1 2.0464,E2 186.1417} C_DIS
LIN {X -23.1572,Y -139.1925,Z 188,A -91.4949,B 2.0519,C 0.272,E1 2.0506,E2 184.6169} C_DIS
LIN {X -18.8262,Y -139.8451,Z 188,A -89.6623,B 2.0519,C 0.272,E1 2.0557,E2 182.7759} C_DIS
LIN {X -15.2921,Y -140.2748,Z 188,A -88.4099,B 2.0517,C 0.2731,E1 2.0591,E2 181.5503} C_DIS
LIN {X -12.132,Y -140.5835,Z 188,A -86.9911,B 2.0518,C 0.2725,E1 2.0631,E2 180.1127} C_DIS
LIN {X -8.77,Y -140.8331,Z 188,A -85.6411,B 2.0518,C 0.2725,E1 2.0669,E2 178.7647} C_DIS
LIN {X -4.8964,Y -141.0222,Z 188,A -84.0213,B 2.0518,C 0.2721,E1 2.0715,E2 177.1378} C_DIS
LIN {X -0.8575,Y -141.1034,Z 188,A -82.3897,B 2.0518,C 0.2719,E1 2.076,E2 175.5067} C_DIS
LIN {X -0.8575,Y -141.1034,Z 188,A -82.3897,B 2.0518,C 0.2719,E1 2.076,E2 175.5067} C_DIS
Enddeposition()
LIN {X 1.0388,Y -141.9991,Z 188,A -81.8394,B 2.0512,C 0.2739,E1 2.077,E2 175.0162} C_DIS
Startdeposition()
$VEL.CP = VEL_PRINT
LIN {X -2.0193,Y -141.9913,Z 188,A -83.5727,B 2.0508,C 0.2768,E1 2.0719,E2 176.8212} C_DIS
LIN {X -6.4778,Y -141.8589,Z 188,A -85.3324,B 2.0508,C 0.2768,E1 2.067,E2 178.5762} C_DIS
LIN {X -10.2141,Y -141.6374,Z 188,A -86.7948,B 2.0508,C 0.2766,E1 2.0629,E2 180.0324} C_DIS
LIN {X -14.1125,Y -141.3032,Z 188,A -88.3488,B 2.0508,C 0.2765,E1 2.0586,E2 181.5836} C_DIS
LIN {X -17.0122,Y -140.9825,Z 188,A -89.5219,B 2.0508,C 0.2763,E1 2.0553,E2 182.7566} C_DIS
LIN {X -20.5487,Y -140.5112,Z 188,A -90.9966,B 2.0508,C 0.2763,E1 2.0512,E2 184.2369} C_DIS
LIN {X -24.1527,Y -139.9382,Z 188,A -92.6075,B 2.0508,C 0.2766,E1 2.0467,E2 185.868} C_DIS
LIN {X -28.4578,Y -139.1243,Z 188,A -94.2767,B 2.0509,C 0.2756,E1 2.0422,E2 187.5238} C_DIS
LIN {X -32.0059,Y -138.3516,Z 188,A -95.8625,B 2.0509,C 0.2756,E1 2.0378,E2 189.1272} C_DIS
LIN {X -36.9658,Y -137.1097,Z 188,A -97.8553,B 2.0511,C 0.2743,E1 2.0324,E2 191.1107} C_DIS
LIN {X -40.1079,Y -136.2233,Z 188,A -99.2237,B 2.0511,C 0.2738,E1 2.0287,E2 192.4868} C_DIS
LIN {X -43.9002,Y -135.0506,Z 188,A -101.225,B 2.0511,C 0.2745,E1 2.0232,E2 194.5449} C_DIS
LIN {X -47.7658,Y -133.7309,Z 188,A -102.3023,B 2.0516,C 0.2709,E1 2.0206,E2 195.5421} C_DIS
LIN {X -50.6603,Y -132.6635,Z 188,A -103.7249,B 2.0516,C 0.2707,E1 2.0168,E2 196.9902} C_DIS
LIN {X -54.1083,Y -131.2938,Z 188,A -105.4038,B 2.0516,C 0.2702,E1 2.0124,E2 198.6951} C_DIS
LIN {X -58.2903,Y -129.4901,Z 188,A -107.1552,B 2.0519,C 0.2681,E1 2.0079,E2 200.4346} C_DIS
LIN {X -61.5858,Y -127.9558,Z 188,A -108.661,B 2.0521,C 0.2668,E1 2.0041,E2 201.9461} C_DIS
LIN {X -64.7591,Y -126.3793,Z 188,A -110.106,B 2.0523,C 0.2654,E1 2.0005,E2 203.3935} C_DIS
LIN {X -67.9097,Y -124.7164,Z 188,A -111.6935,B 2.0524,C 0.2643,E1 1.9965,E2 205.0024} C_DIS
LIN {X -72.0629,Y -122.3636,Z 188,A -113.6682,B 2.0527,C 0.2621,E1 1.9917,E2 206.9842} C_DIS
LIN {X -76.0616,Y -119.9192,Z 188,A -115.6126,B 2.053,C 0.2599,E1 1.987,E2 208.9361} C_DIS
LIN {X -79.9115,Y -117.389,Z 188,A -117.5833,B 2.0533,C 0.2577,E1 1.9824,E2 210.9227} C_DIS
LIN {X -83.6251,Y -114.7731,Z 188,A -119.5399,B 2.0536,C 0.2554,E1 1.9779,E2 212.8967} C_DIS
LIN {X -87.2234,Y -112.0627,Z 188,A -121.3252,B 2.0539,C 0.2525,E1 1.974,E2 214.6774} C_DIS
LIN {X -90.6128,Y -109.3399,Z 188,A -123.1939,B 2.0542,C 0.25,E1 1.9699,E2 216.5621} C_DIS
LIN {X -94.2076,Y -106.2584,Z 188,A -125.1263,B 2.0546,C 0.2469,E1 1.9658,E2 218.4974} C_DIS
LIN {X -97.5166,Y -103.2299,Z 188,A -127.1922,B 2.0549,C 0.2444,E1 1.9615,E2 220.5987} C_DIS
LIN {X -100.6683,Y -100.1589,Z 188,A -128.9068,B 2.0553,C 0.241,E1 1.9581,E2 222.3047} C_DIS
LIN {X -103.8739,Y -96.8303,Z 188,A -130.8191,B 2.0557,C 0.2376,E1 1.9544,E2 224.2235} C_DIS
LIN {X -106.6257,Y -93.7922,Z 188,A -132.7597,B 2.056,C 0.2351,E1 1.9507,E2 226.2036} C_DIS
LIN {X -110.1321,Y -89.6487,Z 188,A -134.8741,B 2.0565,C 0.2304,E1 1.947,E2 228.307} C_DIS
LIN {X -112.8246,Y -86.2352,Z 188,A -137.1007,B 2.0568,C 0.2279,E1 1.9431,E2 230.5983} C_DIS
LIN {X -115.2622,Y -82.9501,Z 188,A -138.5267,B 2.0572,C 0.2237,E1 1.9408,E2 231.9932} C_DIS
LIN {X -117.856,Y -79.2216,Z 188,A -140.4755,B 2.0577,C 0.2199,E1 1.9377,E2 233.9575} C_DIS
LIN {X -121.162,Y -74.0656,Z 188,A -142.7874,B 2.0583,C 0.2139,E1 1.9343,E2 236.2467} C_DIS
LIN {X -122.7018,Y -71.4864,Z 188,A -144.3809,B 2.0585,C 0.2119,E1 1.9319,E2 237.8923} C_DIS
LIN {X -124.9172,Y -67.5406,Z 188,A -146.3114,B 2.0589,C 0.2078,E1 1.9293,E2 239.8365} C_DIS
LIN {X -126.7283,Y -64.0734,Z 188,A -147.8809,B 2.0593,C 0.2039,E1 1.9273,E2 241.4043} C_DIS
LIN {X -128.3525,Y -60.7553,Z 188,A -149.4179,B 2.0597,C 0.2004,E1 1.9254,E2 242.947} C_DIS
LIN {X -129.8763,Y -57.4269,Z 188,A -151.0814,B 2.06,C 0.197,E1 1.9235,E2 244.6354} C_DIS
LIN {X -131.2384,Y -54.2411,Z 188,A -152.4914,B 2.0603,C 0.1935,E1 1.922,E2 246.0465} C_DIS
LIN {X -132.6364,Y -50.7299,Z 188,A -154.2589,B 2.0606,C 0.1901,E1 1.9201,E2 247.8463} C_DIS
LIN {X -134.2501,Y -46.2853,Z 188,A -156.2091,B 2.0611,C 0.1852,E1 1.9183,E2 249.8014} C_DIS
LIN {X -135.4795,Y -42.5576,Z 188,A -157.8753,B 2.0614,C 0.1812,E1 1.9169,E2 251.4782} C_DIS
LIN {X -136.3827,Y -39.5633,Z 188,A -159.2151,B 2.0617,C 0.1779,E1 1.9158,E2 252.8278} C_DIS
LIN {X -137.2517,Y -36.4332,Z 188,A -160.704,B 2.062,C 0.1748,E1 1.9147,E2 254.34} C_DIS
LIN {X -138.2703,Y -32.3619,Z 188,A -162.6037,B 2.0623,C 0.1705,E1 1.9134,E2 256.2667} C_DIS
LIN {X -139.6261,Y -25.8956,Z 188,A -166.21,B 2.0628,C 0.1648,E1 1.9114,E2 259.9966} C_DIS
LIN {X -140.6377,Y -19.6632,Z 188,A -167.9394,B 2.0635,C 0.1564,E1 1.9108,E2 261.616} C_DIS
LIN {X -140.9993,Y -16.871,Z 188,A -169.2895,B 2.0637,C 0.1536,E1 1.9103,E2 262.9941} C_DIS
LIN {X -141.3505,Y -13.6193,Z 188,A -170.7409,B 2.0639,C 0.1502,E1 1.9099,E2 264.4623} C_DIS
LIN {X -141.7589,Y -8.3674,Z 188,A -173.0413,B 2.0643,C 0.1445,E1 1.9094,E2 266.7846} C_DIS
LIN {X -141.9325,Y -4.5886,Z 188,A -174.7257,B 2.0646,C 0.1405,E1 1.9092,E2 268.4891} C_DIS
LIN {X -142.0061,Y -0.436,Z 188,A -176.4266,B 2.0649,C 0.1358,E1 1.9092,E2 270.1924} C_DIS
LIN {X -141.9578,Y 3.6786,Z 188,A -178.3119,B 2.0652,C 0.1315,E1 1.9092,E2 272.1062} C_DIS
LIN {X -141.7417,Y 8.6471,Z 188,A 179.5644,B 2.0655,C 0.1261,E1 1.9096,E2 274.2439} C_DIS
LIN {X -141.4438,Y 12.6317,Z 188,A 177.8518,B 2.0658,C 0.1218,E1 1.91,E2 275.9688} C_DIS
LIN {X -140.9367,Y 17.3963,Z 188,A 175.8489,B 2.0661,C 0.1165,E1 1.9106,E2 277.9796} C_DIS
LIN {X -140.4311,Y 21.0937,Z 188,A 173.7253,B 2.0663,C 0.1133,E1 1.9115,E2 280.1824} C_DIS
LIN {X -139.7386,Y 25.2705,Z 188,A 172.8229,B 2.0666,C 0.1073,E1 1.9119,E2 280.9788} C_DIS
LIN {X -138.4456,Y 31.5943,Z 188,A 169.7936,B 2.0669,C 0.1009,E1 1.9136,E2 284.0621} C_DIS
LIN {X -136.8865,Y 37.7849,Z 188,A 166.9866,B 2.0672,C 0.0943,E1 1.9156,E2 286.8975} C_DIS
LIN {X -136.1225,Y 40.452,Z 188,A 165.6482,B 2.0673,C 0.0916,E1 1.9166,E2 288.2635} C_DIS
LIN {X -135.1987,Y 43.4364,Z 188,A 164.2316,B 2.0675,C 0.0885,E1 1.9178,E2 289.6992} C_DIS
LIN {X -134.0537,Y 46.8518,Z 188,A 162.7377,B 2.0676,C 0.0847,E1 1.9192,E2 291.1973} C_DIS
LIN {X -132.6884,Y 50.5947,Z 188,A 161.0108,B 2.0678,C 0.0808,E1 1.9209,E2 292.9385} C_DIS
LIN {X -131.2111,Y 54.3065,Z 188,A 159.0764,B 2.0679,C 0.0772,E1 1.923,E2 294.9129} C_DIS
LIN {X -129.3131,Y 58.6859,Z 188,A 156.5964,B 2.0681,C 0.0733,E1 1.9259,E2 297.4619} C_DIS
LIN {X -127.1721,Y 63.1881,Z 188,A 155.0652,B 2.0683,C 0.0674,E1 1.9277,E2 298.9307} C_DIS
LIN {X -125.3768,Y 66.6822,Z 188,A 153.3186,B 2.0683,C 0.0638,E1 1.93,E2 300.6968} C_DIS
LIN {X -122.8469,Y 71.2358,Z 188,A 151.1996,B 2.0685,C 0.0588,E1 1.9329,E2 302.8164} C_DIS
LIN {X -120.8995,Y 74.4936,Z 188,A 149.4407,B 2.0686,C 0.0557,E1 1.9355,E2 304.6031} C_DIS
LIN {X -118.5242,Y 78.2172,Z 188,A 147.5619,B 2.0687,C 0.0518,E1 1.9384,E2 306.4928} C_DIS
LIN {X -115.8609,Y 82.1112,Z 188,A 145.446,B 2.0688,C 0.0479,E1 1.9418,E2 308.6341} C_DIS
LIN {X -112.425,Y 86.756,Z 188,A 143.0922,B 2.0689,C 0.0429,E1 1.9457,E2 310.9889} C_DIS
LIN {X -109.6385,Y 90.2522,Z 188,A 141.2204,B 2.069,C 0.0393,E1 1.949,E2 312.8681} C_DIS
LIN {X -106.8258,Y 93.5639,Z 188,A 139.3639,B 2.069,C 0.0359,E1 1.9525,E2 314.7362} C_DIS
LIN {X -103.8627,Y 96.8423,Z 188,A 137.4577,B 2.0691,C 0.0327,E1 1.9561,E2 316.6565} C_DIS
LIN {X -100.5903,Y 100.2373,Z 188,A 135.4666,B 2.0691,C 0.0293,E1 1.96,E2 318.6572} C_DIS
LIN {X -97.238,Y 103.4927,Z 188,A 133.4856,B 2.0692,C 0.0261,E1 1.964,E2 320.6488} C_DIS
LIN {X -93.8243,Y 106.5973,Z 188,A 131.5341,B 2.0692,C 0.023,E1 1.9681,E2 322.6102} C_DIS
LIN {X -90.2597,Y 109.6323,Z 188,A 129.5382,B 2.0692,C 0.0201,E1 1.9724,E2 324.6181} C_DIS
LIN {X -86.7167,Y 112.4555,Z 188,A 127.7046,B 2.0693,C 0.0172,E1 1.9765,E2 326.4511} C_DIS
LIN {X -83.1399,Y 115.1247,Z 188,A 125.681,B 2.0693,C 0.0151,E1 1.9811,E2 328.501} C_DIS
LIN {X -78.9532,Y 118.0352,Z 188,A 123.7167,B 2.0693,C 0.0118,E1 1.9856,E2 330.4524} C_DIS
LIN {X -75.4268,Y 120.3199,Z 188,A 121.8772,B 2.0693,C 0.0099,E1 1.99,E2 332.3086} C_DIS
LIN {X -71.5431,Y 122.669,Z 188,A 120.018,B 2.0693,C 0.0077,E1 1.9944,E2 334.1701} C_DIS
LIN {X -67.2619,Y 125.0669,Z 188,A 118.0314,B 2.0693,C 0.0053,E1 1.9993,E2 336.1561} C_DIS
LIN {X -63.8965,Y 126.8184,Z 188,A 116.4687,B 2.0693,C 0.0037,E1 2.0032,E2 337.7218} C_DIS
LIN {X -60.1574,Y 128.6343,Z 188,A 114.7094,B 2.0693,C 0.0022,E1 2.0077,E2 339.4902} C_DIS
LIN {X -57.3971,Y 129.8896,Z 188,A 113.5221,B 2.0693,C 0.0009,E1 2.0107,E2 340.6723} C_DIS
LIN {X -54.1567,Y 131.2736,Z 188,A 112.096,B 2.0693,C -0.0004,E1 2.0144,E2 342.0982} C_DIS
LIN {X -51.364,Y 132.3899,Z 188,A 110.7829,B 2.0693,C -0.001,E1 2.0178,E2 343.4226} C_DIS
LIN {X -47.5661,Y 133.8029,Z 188,A 109.1471,B 2.0693,C -0.0023,E1 2.0221,E2 345.0577} C_DIS
LIN {X -44.3592,Y 134.8996,Z 188,A 107.7899,B 2.0693,C -0.0033,E1 2.0257,E2 346.4128} C_DIS
LIN {X -41.2358,Y 135.8863,Z 188,A 106.4291,B 2.0693,C -0.004,E1 2.0294,E2 347.7776} C_DIS
LIN {X -38.0621,Y 136.809,Z 188,A 104.9824,B 2.0693,C -0.0044,E1 2.0333,E2 349.2374} C_DIS
LIN {X -34.3526,Y 137.7884,Z 188,A 103.5309,B 2.0693,C -0.0055,E1 2.0372,E2 350.6763} C_DIS
LIN {X -31.739,Y 138.4126,Z 188,A 102.4198,B 2.0693,C -0.0059,E1 2.0403,E2 351.7901} C_DIS
LIN {X -27.7196,Y 139.2745,Z 188,A 100.752,B 2.0693,C -0.0065,E1 2.0448,E2 353.4583} C_DIS
LIN {X -25.0019,Y 139.7867,Z 188,A 99.5362,B 2.0693,C -0.0065,E1 2.0482,E2 354.6856} C_DIS
LIN {X -21.0665,Y 140.4353,Z 188,A 97.8672,B 2.0693,C -0.0065,E1 2.0529,E2 356.3613} C_DIS
LIN {X -16.397,Y 141.0559,Z 188,A 96.1042,B 2.0693,C -0.0074,E1 2.0577,E2 358.1065} C_DIS
LIN {X -12.4883,Y 141.456,Z 188,A 94.3826,B 2.0693,C -0.0069,E1 2.0625,E2 359.844} C_DIS
LIN {X -8.1462,Y 141.7725,Z 188,A 92.768,B 2.0693,C -0.0075,E1 2.067,E2 361.4405} C_DIS
LIN {X -4.8457,Y 141.9242,Z 188,A 91.4327,B 2.0693,C -0.0075,E1 2.0707,E2 362.7756} C_DIS
LIN {X -1.5849,Y 141.9985,Z 188,A 89.972,B 2.0693,C -0.0065,E1 2.0749,E2 364.2534} C_DIS
LIN {X 3.0542,Y 141.9741,Z 188,A 88.2601,B 2.0693,C -0.0069,E1 2.0796,E2 365.9449} C_DIS
LIN {X 6.0378,Y 141.8777,Z 188,A 87.0437,B 2.0693,C -0.0064,E1 2.083,E2 367.1624} C_DIS
LIN {X 10.4915,Y 141.6171,Z 188,A 85.233,B 2.0693,C -0.0057,E1 2.0881,E2 368.9737} C_DIS
LIN {X 13.5445,Y 141.3577,Z 188,A 84.0322,B 2.0693,C -0.0053,E1 2.0914,E2 370.1697} C_DIS
LIN {X 17.1598,Y 140.9649,Z 188,A 82.6202,B 2.0693,C -0.0048,E1 2.0953,E2 371.5744} C_DIS
LIN {X 20.3939,Y 140.5333,Z 188,A 81.2876,B 2.0693,C -0.004,E1 2.099,E2 372.9086} C_DIS
LIN {X 24.3343,Y 139.9062,Z 188,A 79.7188,B 2.0693,C -0.0031,E1 2.1034,E2 374.4719} C_DIS
LIN {X 27.2631,Y 139.3646,Z 188,A 78.3971,B 2.0693,C -0.0016,E1 2.107,E2 375.8079} C_DIS
LIN {X 32.0104,Y 138.3506,Z 188,A 76.5869,B 2.0693,C -0.0009,E1 2.1119,E2 377.5993} C_DIS
LIN {X 35.5931,Y 137.4736,Z 188,A 75.162,B 2.0693,C 0.0001,E1 2.1158,E2 379.0161} C_DIS
LIN {X 38.7398,Y 136.6194,Z 188,A 73.9078,B 2.0693,C 0.001,E1 2.1191,E2 380.2624} C_DIS
LIN {X 44.0229,Y 135.0114,Z 188,A 71.6814,B 2.0693,C 0.0032,E1 2.1251,E2 382.4882} C_DIS
LIN {X 46.9133,Y 134.0324,Z 188,A 70.3725,B 2.0693,C 0.005,E1 2.1286,E2 383.8063} C_DIS
LIN {X 51.2129,Y 132.4487,Z 188,A 68.5885,B 2.0693,C 0.0068,E1 2.1332,E2 385.5819} C_DIS
LIN {X 55.3149,Y 130.7899,Z 188,A 66.9389,B 2.0693,C 0.0082,E1 2.1374,E2 387.2146} C_DIS
LIN {X 58.3655,Y 129.4565,Z 188,A 65.6204,B 2.0693,C 0.0098,E1 2.1408,E2 388.5297} C_DIS
LIN {X 61.5585,Y 127.9688,Z 188,A 64.2565,B 2.0693,C 0.0114,E1 2.1442,E2 389.8864} C_DIS
LIN {X 64.8345,Y 126.3409,Z 188,A 62.8193,B 2.0693,C 0.0132,E1 2.1478,E2 391.3186} C_DIS
LIN {X 68.4861,Y 124.4013,Z 188,A 61.1302,B 2.0693,C 0.0158,E1 2.152,E2 393.0102} C_DIS
LIN {X 72.4702,Y 122.1231,Z 188,A 59.3907,B 2.0693,C 0.018,E1 2.1562,E2 394.7357} C_DIS
LIN {X 76.0662,Y 119.9163,Z 188,A 57.7151,B 2.0693,C 0.0206,E1 2.1601,E2 396.4078} C_DIS
LIN {X 79.961,Y 117.3555,Z 188,A 55.8999,B 2.0693,C 0.0234,E1 2.1643,E2 398.2149} C_DIS
LIN {X 83.8132,Y 114.6357,Z 188,A 54.2129,B 2.0693,C 0.0253,E1 2.1681,E2 399.8749} C_DIS
LIN {X 86.7967,Y 112.3935,Z 188,A 52.6992,B 2.0692,C 0.0281,E1 2.1715,E2 401.3896} C_DIS
LIN {X 90.2059,Y 109.6767,Z 188,A 50.9457,B 2.0692,C 0.0314,E1 2.1753,E2 403.1426} C_DIS
LIN {X 93.6457,Y 106.7544,Z 188,A 49.2734,B 2.0691,C 0.0339,E1 2.1788,E2 404.7962} C_DIS
LIN {X 97.0035,Y 103.7126,Z 188,A 47.5891,B 2.0691,C 0.0366,E1 2.1822,E2 406.4626} C_DIS
LIN {X 99.8283,Y 100.9967,Z 188,A 46.0132,B 2.069,C 0.0398,E1 2.1854,E2 408.038} C_DIS
LIN {X 102.6439,Y 98.1332,Z 188,A 44.4518,B 2.069,C 0.0428,E1 2.1884,E2 409.5922} C_DIS
LIN {X 105.7257,Y 94.8049,Z 188,A 42.714,B 2.0689,C 0.0461,E1 2.1917,E2 411.3186} C_DIS
LIN {X 108.6674,Y 91.4184,Z 188,A 41.0002,B 2.0688,C 0.0495,E1 2.1948,E2 413.0205} C_DIS
LIN {X 111.4637,Y 87.9879,Z 188,A 39.1837,B 2.0687,C 0.0537,E1 2.1979,E2 414.8413} C_DIS
LIN {X 114.6196,Y 83.8352,Z 188,A 37.3144,B 2.0686,C 0.0569,E1 2.201,E2 416.6811} C_DIS
LIN {X 116.9906,Y 80.493,Z 188,A 35.7539,B 2.0686,C 0.0601,E1 2.2035,E2 418.2302} C_DIS
LIN {X 119.5728,Y 76.6044,Z 188,A 34.1051,B 2.0684,C 0.063,E1 2.206,E2 419.8495} C_DIS
LIN {X 121.6456,Y 73.2688,Z 188,A 32.4597,B 2.0683,C 0.0673,E1 2.2084,E2 421.5031} C_DIS
LIN {X 123.8447,Y 69.4866,Z 188,A 30.8296,B 2.0682,C 0.0707,E1 2.2106,E2 423.1165} C_DIS
LIN {X 125.9292,Y 65.6304,Z 188,A 29.214,B 2.0681,C 0.074,E1 2.2127,E2 424.7128} C_DIS
LIN {X 127.5041,Y 62.515,Z 188,A 27.8861,B 2.0679,C 0.077,E1 2.2144,E2 426.0309} C_DIS
LIN {X 129.0824,Y 59.1885,Z 188,A 26.4771,B 2.0679,C 0.0802,E1 2.216,E2 427.4304} C_DIS
LIN {X 130.7824,Y 55.3329,Z 188,A 24.7737,B 2.0676,C 0.0847,E1 2.2179,E2 429.135} C_DIS
LIN {X 132.4116,Y 51.3082,Z 188,A 23.2235,B 2.0676,C 0.0877,E1 2.2195,E2 430.6596} C_DIS
LIN {X 133.7026,Y 47.8443,Z 188,A 21.8486,B 2.0674,C 0.0908,E1 2.2208,E2 432.02} C_DIS
LIN {X 134.905,Y 44.3429,Z 188,A 20.3291,B 2.0672,C 0.095,E1 2.2221,E2 433.5435} C_DIS
LIN {X 136.5936,Y 38.8323,Z 188,A 18.3555,B 2.067,C 0.0986,E1 2.2237,E2 435.4723} C_DIS
LIN {X 137.889,Y 33.9485,Z 188,A 16.2765,B 2.0667,C 0.1044,E1 2.2251,E2 437.5575} C_DIS
LIN {X 139.0962,Y 28.596,Z 188,A 14.475,B 2.0666,C 0.1073,E1 2.2262,E2 439.306} C_DIS
LIN {X 139.538,Y 26.3562,Z 188,A 13.4768,B 2.0664,C 0.1105,E1 2.2267,E2 440.3148} C_DIS
LIN {X 140.0872,Y 23.2593,Z 188,A 12.1829,B 2.0662,C 0.1142,E1 2.2273,E2 441.6126} C_DIS
LIN {X 140.6933,Y 19.2742,Z 188,A 10.7227,B 2.066,C 0.1174,E1 2.2279,E2 443.0519} C_DIS
LIN {X 141.1296,Y 15.7543,Z 188,A 9.2593,B 2.0658,C 0.1216,E1 2.2284,E2 444.5203} C_DIS
LIN {X 141.5114,Y 11.8322,Z 188,A 7.8669,B 2.0656,C 0.1245,E1 2.2287,E2 445.8874} C_DIS
LIN {X 141.7666,Y 8.2426,Z 188,A 6.5806,B 2.0655,C 0.1273,E1 2.229,E2 447.1526} C_DIS
LIN {X 141.9091,Y 5.2328,Z 188,A 5.4156,B 2.0653,C 0.1303,E1 2.2291,E2 448.3115} C_DIS
LIN {X 141.9874,Y 2.2519,Z 188,A 4.2565,B 2.0651,C 0.1333,E1 2.2291,E2 449.4655} C_DIS
LIN {X 141.9885,Y -2.1888,Z 188,A 2.5158,B 2.0648,C 0.1379,E1 2.2291,E2 451.2005} C_DIS
LIN {X 141.8992,Y -5.4858,Z 188,A 1.2954,B 2.0646,C 0.1408,E1 2.2291,E2 452.407} C_DIS
LIN {X 141.6601,Y -9.903,Z 188,A -0.3776,B 2.0643,C 0.1449,E1 2.2288,E2 454.0661} C_DIS
LIN {X 141.2834,Y -14.3189,Z 188,A -1.9871,B 2.064,C 0.1485,E1 2.2284,E2 455.653} C_DIS
LIN {X 140.9405,Y -17.3639,Z 188,A -3.2005,B 2.0638,C 0.1518,E1 2.228,E2 456.864} C_DIS
LIN {X 140.3362,Y -21.7069,Z 188,A -4.9033,B 2.0635,C 0.1562,E1 2.2273,E2 458.559} C_DIS
LIN {X 139.7169,Y -25.3917,Z 188,A -6.2373,B 2.0633,C 0.159,E1 2.2266,E2 459.8707} C_DIS
LIN {X 138.923,Y -29.4295,Z 188,A -7.7005,B 2.063,C 0.162,E1 2.2258,E2 461.3085} C_DIS
LIN {X 138.2297,Y -32.5349,Z 188,A -8.9681,B 2.0628,C 0.1654,E1 2.2251,E2 462.5748} C_DIS
LIN {X 137.6279,Y -34.985,Z 188,A -10.0154,B 2.0625,C 0.1684,E1 2.2243,E2 463.6268} C_DIS
LIN {X 136.6966,Y -38.4637,Z 188,A -11.3329,B 2.0623,C 0.1713,E1 2.2234,E2 464.9268} C_DIS
LIN {X 134.0945,Y -46.7341,Z 188,A -14.6252,B 2.0616,C 0.1791,E1 2.2206,E2 468.1938} C_DIS
LIN {X 132.6665,Y -50.6525,Z 188,A -16.1811,B 2.0613,C 0.1825,E1 2.2191,E2 469.7337} C_DIS
LIN {X 131.189,Y -54.3593,Z 188,A -17.8206,B 2.0609,C 0.187,E1 2.2174,E2 471.3784} C_DIS
LIN {X 129.3319,Y -58.644,Z 188,A -19.4627,B 2.0606,C 0.19,E1 2.2155,E2 472.9888} C_DIS
LIN {X 127.2027,Y -63.1261,Z 188,A -21.3621,B 2.0602,C 0.1944,E1 2.2133,E2 474.8757} C_DIS
LIN {X 125.5362,Y -66.3787,Z 188,A -22.6956,B 2.06,C 0.197,E1 2.2116,E2 476.191} C_DIS
LIN {X 123.6569,Y -69.8208,Z 188,A -24.5534,B 2.0594,C 0.2031,E1 2.209,E2 478.0879} C_DIS
LIN {X 121.824,Y -72.9716,Z 188,A -25.804,B 2.0592,C 0.205,E1 2.2072,E2 479.3094} C_DIS
LIN {X 119.1209,Y -77.3053,Z 188,A -27.6353,B 2.0589,C 0.2083,E1 2.2045,E2 481.1107} C_DIS
LIN {X 116.783,Y -80.7946,Z 188,A -29.262,B 2.0585,C 0.2118,E1 2.202,E2 482.7293} C_DIS
LIN {X 114.1748,Y -84.4406,Z 188,A -31.0024,B 2.0581,C 0.2155,E1 2.1991,E2 484.4617} C_DIS
LIN {X 111.3476,Y -88.1348,Z 188,A -32.7677,B 2.0578,C 0.219,E1 2.1961,E2 486.213} C_DIS
LIN {X 108.4059,Y -91.7287,Z 188,A -34.5433,B 2.0574,C 0.2225,E1 2.193,E2 487.9765} C_DIS
LIN {X 105.4516,Y -95.1106,Z 188,A -36.274,B 2.057,C 0.2258,E1 2.1898,E2 489.6973} C_DIS
LIN {X 102.2668,Y -98.5268,Z 188,A -38.007,B 2.0567,C 0.2287,E1 2.1865,E2 491.4108} C_DIS
LIN {X 99.1653,Y -101.6478,Z 188,A -39.7255,B 2.0563,C 0.232,E1 2.1831,E2 493.1227} C_DIS
LIN {X 95.8278,Y -104.8001,Z 188,A -41.5005,B 2.056,C 0.2352,E1 2.1795,E2 494.8883} C_DIS
LIN {X 92.3605,Y -107.8684,Z 188,A -43.2954,B 2.0556,C 0.2384,E1 2.1757,E2 496.6745} C_DIS
LIN {X 88.7764,Y -110.837,Z 188,A -45.0917,B 2.0553,C 0.2414,E1 2.1718,E2 498.4609} C_DIS
LIN {X 85.2825,Y -113.5469,Z 188,A -46.7323,B 2.055,C 0.2436,E1 2.1682,E2 500.0826} C_DIS
LIN {X 81.8198,Y -116.0664,Z 188,A -48.4112,B 2.0547,C 0.2463,E1 2.1644,E2 501.756} C_DIS
LIN {X 78.1416,Y -118.574,Z 188,A -50.1414,B 2.0543,C 0.249,E1 2.1604,E2 503.4783} C_DIS
LIN {X 74.5598,Y -120.8589,Z 188,A -51.8379,B 2.054,C 0.2517,E1 2.1564,E2 505.1736} C_DIS
LIN {X 70.7248,Y -123.1425,Z 188,A -53.5479,B 2.0537,C 0.2539,E1 2.1523,E2 506.8722} C_DIS
LIN {X 66.2016,Y -125.6292,Z 188,A -55.2338,B 2.0537,C 0.2544,E1 2.1483,E2 508.5035} C_DIS
LIN {X 64.0775,Y -126.7262,Z 188,A -56.42,B 2.0533,C 0.2572,E1 2.1453,E2 509.7218} C_DIS
LIN {X 60.4458,Y -128.5004,Z 188,A -58.0732,B 2.053,C 0.2597,E1 2.1411,E2 511.3793} C_DIS
LIN {X 55.1119,Y -130.8747,Z 188,A -60.0969,B 2.053,C 0.2606,E1 2.136,E2 513.3578} C_DIS
LIN {X 51.026,Y -132.5213,Z 188,A -61.9599,B 2.0526,C 0.2633,E1 2.1311,E2 515.2341} C_DIS
LIN {X 48.1289,Y -133.6,Z 188,A -63.2215,B 2.0524,C 0.2649,E1 2.1278,E2 516.4985} C_DIS
LIN {X 44.2008,Y -134.9523,Z 188,A -65.1682,B 2.0519,C 0.2684,E1 2.1225,E2 518.4846} C_DIS
LIN {X 40.6059,Y -136.0775,Z 188,A -66.2583,B 2.052,C 0.2673,E1 2.1198,E2 519.5149} C_DIS
LIN {X 36.29,Y -137.2899,Z 188,A -68.0823,B 2.0518,C 0.2691,E1 2.1148,E2 521.3422} C_DIS
LIN {X 32.4653,Y -138.2465,Z 188,A -70.0374,B 2.0513,C 0.2727,E1 2.1094,E2 523.3499} C_DIS
LIN {X 28.613,Y -139.0928,Z 188,A -71.34,B 2.0514,C 0.2722,E1 2.1059,E2 524.6126} C_DIS
LIN {X 24.2878,Y -139.9145,Z 188,A -72.9187,B 2.0514,C 0.2723,E1 2.1016,E2 526.1645} C_DIS
LIN {X 20.7906,Y -140.4766,Z 188,A -74.4469,B 2.0512,C 0.2738,E1 2.0974,E2 527.7075} C_DIS
LIN {X 16.5984,Y -141.0319,Z 188,A -76.0448,B 2.0512,C 0.2742,E1 2.093,E2 529.291} C_DIS
LIN {X 13.2179,Y -141.3891,Z 188,A -77.319,B 2.0512,C 0.2743,E1 2.0894,E2 530.5521} C_DIS
LIN {X 10.2672,Y -141.6335,Z 188,A -78.5314,B 2.051,C 0.2749,E1 2.086,E2 531.7677} C_DIS
LIN {X 6.5308,Y -141.8562,Z 188,A -80.1864,B 2.0509,C 0.2763,E1 2.0814,E2 533.444} C_DIS
LIN {X 2.2633,Y -141.9872,Z 188,A -81.7769,B 2.0509,C 0.2761,E1 2.077,E2 535.0166} C_DIS
LIN {X 2.2633,Y -141.9872,Z 188,A -81.7769,B 2.0509,C 0.2761,E1 2.077,E2 535.0166} C_DIS
Enddeposition()
LIN {X 1.0451,Y -142.9001,Z 188,A -81.9413,B 2.0509,C 0.2755,E1 2.0765,E2 535.1638} C_DIS
Startdeposition()
$VEL.CP = VEL_PRINT
LIN {X 3.5139,Y -142.8621,Z 188,A -80.6297,B 2.0512,C 0.2735,E1 2.0803,E2 533.8053} C_DIS
LIN {X 7.0145,Y -142.7323,Z 188,A -79.2463,B 2.0512,C 0.2731,E1 2.0841,E2 532.4242} C_DIS
LIN {X 10.5108,Y -142.5174,Z 188,A -77.8147,B 2.0513,C 0.2724,E1 2.0881,E2 530.988} C_DIS
LIN {X 14.3724,Y -142.1817,Z 188,A -76.3473,B 2.0513,C 0.2721,E1 2.0922,E2 529.5323} C_DIS
LIN {X 17.6196,Y -141.8157,Z 188,A -75.0471,B 2.0514,C 0.2714,E1 2.0958,E2 528.2328} C_DIS
LIN {X 21.4252,Y -141.2898,Z 188,A -73.6545,B 2.0514,C 0.2714,E1 2.0996,E2 526.8606} C_DIS
LIN {X 24.4316,Y -140.8024,Z 188,A -72.2865,B 2.0517,C 0.2696,E1 2.1035,E2 525.4708} C_DIS
LIN {X 27.9283,Y -140.1498,Z 188,A -70.906,B 2.0517,C 0.2688,E1 2.1072,E2 524.0959} C_DIS
LIN {X 31.3498,Y -139.424,Z 188,A -69.5336,B 2.0519,C 0.2679,E1 2.111,E2 522.727} C_DIS
LIN {X 35.1838,Y -138.5053,Z 188,A -68.088,B 2.0519,C 0.2673,E1 2.1149,E2 521.2999} C_DIS
LIN {X 38.1169,Y -137.7275,Z 188,A -66.8002,B 2.0522,C 0.2657,E1 2.1184,E2 520.001} C_DIS
LIN {X 41.4643,Y -136.7569,Z 188,A -65.4365,B 2.0523,C 0.2645,E1 2.122,E2 518.6414} C_DIS
LIN {X 44.8334,Y -135.6896,Z 188,A -64.0542,B 2.0525,C 0.2632,E1 2.1257,E2 517.2631} C_DIS
LIN {X 48.5757,Y -134.3949,Z 188,A -62.6012,B 2.0526,C 0.2623,E1 2.1295,E2 515.8283} C_DIS
LIN {X 51.4298,Y -133.3292,Z 188,A -61.3205,B 2.0528,C 0.2605,E1 2.1329,E2 514.5383} C_DIS
LIN {X 54.7251,Y -132.0109,Z 188,A -59.9438,B 2.053,C 0.259,E1 2.1364,E2 513.1672} C_DIS
LIN {X 58.1468,Y -130.5395,Z 188,A -58.5543,B 2.0532,C 0.2577,E1 2.1399,E2 511.7916} C_DIS
LIN {X 61.115,Y -129.1774,Z 188,A -57.2327,B 2.0534,C 0.2559,E1 2.1433,E2 510.4675} C_DIS
LIN {X 64.2541,Y -127.6455,Z 188,A -55.8187,B 2.0537,C 0.2538,E1 2.1469,E2 509.0505} C_DIS
LIN {X 67.947,Y -125.7198,Z 188,A -54.2243,B 2.0539,C 0.2518,E1 2.1508,E2 507.4657} C_DIS
LIN {X 71.7677,Y -123.5782,Z 188,A -52.5378,B 2.0542,C 0.2496,E1 2.1549,E2 505.788} C_DIS
LIN {X 75.1646,Y -121.5424,Z 188,A -50.9233,B 2.0545,C 0.2468,E1 2.1587,E2 504.1684} C_DIS
LIN {X 78.8532,Y -119.1822,Z 188,A -49.2383,B 2.0548,C 0.2443,E1 2.1626,E2 502.4923} C_DIS
LIN {X 82.8097,Y -116.4681,Z 188,A -47.4187,B 2.0551,C 0.2417,E1 2.1668,E2 500.6861} C_DIS
LIN {X 86.5342,Y -113.7281,Z 188,A -45.6189,B 2.0555,C 0.2387,E1 2.1708,E2 498.8927} C_DIS
LIN {X 90.1569,Y -110.8782,Z 188,A -43.8517,B 2.0558,C 0.2358,E1 2.1746,E2 497.1356} C_DIS
LIN {X 93.5127,Y -108.063,Z 188,A -42.1707,B 2.0561,C 0.2329,E1 2.1782,E2 495.4639} C_DIS
LIN {X 97.0977,Y -104.8538,Z 188,A -40.403,B 2.0565,C 0.2303,E1 2.1818,E2 493.7177} C_DIS
LIN {X 99.9669,Y -102.1213,Z 188,A -38.8386,B 2.0568,C 0.2272,E1 2.1849,E2 492.1554} C_DIS
LIN {X 103.0506,Y -99.0092,Z 188,A -37.1493,B 2.0571,C 0.224,E1 2.1882,E2 490.4744} C_DIS
LIN {X 106.045,Y -95.795,Z 188,A -35.5201,B 2.0575,C 0.2211,E1 2.1913,E2 488.8625} C_DIS
LIN {X 108.9313,Y -92.4992,Z 188,A -33.8665,B 2.0578,C 0.218,E1 2.1943,E2 487.2221} C_DIS
LIN {X 111.7149,Y -89.1175,Z 188,A -32.1614,B 2.0582,C 0.2144,E1 2.1973,E2 485.5229} C_DIS
LIN {X 114.2672,Y -85.821,Z 188,A -30.6467,B 2.0584,C 0.2118,E1 2.1998,E2 484.029} C_DIS
LIN {X 116.8429,Y -82.2793,Z 188,A -28.982,B 2.0588,C 0.2083,E1 2.2025,E2 482.3757} C_DIS
LIN {X 119.1826,Y -78.8527,Z 188,A -27.3988,B 2.0591,C 0.205,E1 2.2049,E2 480.8026} C_DIS
LIN {X 121.2282,Y -75.6695,Z 188,A -25.9701,B 2.0594,C 0.202,E1 2.207,E2 479.3851} C_DIS
LIN {X 123.4862,Y -71.9265,Z 188,A -24.3117,B 2.0598,C 0.1984,E1 2.2094,E2 477.7386} C_DIS
LIN {X 125.6262,Y -68.1198,Z 188,A -22.6406,B 2.0601,C 0.1946,E1 2.2116,E2 476.0774} C_DIS
LIN {X 127.2503,Y -65.0303,Z 188,A -21.392,B 2.0604,C 0.1922,E1 2.2132,E2 474.8488} C_DIS
LIN {X 128.7981,Y -61.9089,Z 188,A -20.0687,B 2.0606,C 0.1892,E1 2.2148,E2 473.5347} C_DIS
LIN {X 130.2877,Y -58.7096,Z 188,A -18.6604,B 2.061,C 0.1856,E1 2.2165,E2 472.1262} C_DIS
LIN {X 132.0288,Y -54.682,Z 188,A -17.0523,B 2.0613,C 0.1822,E1 2.2182,E2 470.5378} C_DIS
LIN {X 133.4948,Y -51.0039,Z 188,A -15.5982,B 2.0615,C 0.1791,E1 2.2196,E2 469.1012} C_DIS
LIN {X 134.5496,Y -48.1465,Z 188,A -14.406,B 2.0618,C 0.1761,E1 2.2208,E2 467.9121} C_DIS
LIN {X 135.8528,Y -44.3433,Z 188,A -12.9341,B 2.0621,C 0.1729,E1 2.2221,E2 466.4585} C_DIS
LIN {X 137.0357,Y -40.5336,Z 188,A -11.4156,B 2.0624,C 0.1692,E1 2.2233,E2 464.9499} C_DIS
LIN {X 137.8552,Y -37.6599,Z 188,A -10.3148,B 2.0626,C 0.1667,E1 2.2241,E2 463.8617} C_DIS
LIN {X 138.6271,Y -34.7037,Z 188,A -9.1133,B 2.0628,C 0.1635,E1 2.2249,E2 462.6626} C_DIS
LIN {X 139.5351,Y -30.8561,Z 188,A -7.6668,B 2.0631,C 0.1603,E1 2.2258,E2 461.2341} C_DIS
LIN {X 140.249,Y -27.4268,Z 188,A -6.3503,B 2.0633,C 0.1571,E1 2.2265,E2 459.9287} C_DIS
LIN {X 140.8784,Y -23.982,Z 188,A -5.1734,B 2.0635,C 0.1551,E1 2.2271,E2 458.782} C_DIS
LIN {X 141.4233,Y -20.5234,Z 188,A -3.7194,B 2.0638,C 0.1508,E1 2.2277,E2 457.3201} C_DIS
LIN {X 141.885,Y -17.039,Z 188,A -2.4033,B 2.064,C 0.1476,E1 2.2282,E2 456.0159} C_DIS
LIN {X 142.2174,Y -14.0002,Z 188,A -1.2521,B 2.0642,C 0.1447,E1 2.2285,E2 454.8741} C_DIS
LIN {X 142.5507,Y -10.0556,Z 188,A 0.1685,B 2.0644,C 0.1416,E1 2.2288,E2 453.4752} C_DIS
LIN {X 142.7553,Y -6.5582,Z 188,A 1.5248,B 2.0647,C 0.1381,E1 2.229,E2 452.1246} C_DIS
LIN {X 142.8819,Y -2.5509,Z 188,A 3.0979,B 2.065,C 0.1339,E1 2.2291,E2 450.5552} C_DIS
LIN {X 142.8951,Y 1.7582,Z 188,A 4.6833,B 2.0652,C 0.1302,E1 2.2291,E2 448.988} C_DIS
LIN {X 142.808,Y 5.26,Z 188,A 5.9886,B 2.0654,C 0.127,E1 2.229,E2 447.6953} C_DIS
LIN {X 142.6359,Y 8.7581,Z 188,A 7.3312,B 2.0656,C 0.1236,E1 2.2288,E2 446.3602} C_DIS
LIN {X 142.3385,Y 12.725,Z 188,A 8.7617,B 2.0658,C 0.1204,E1 2.2284,E2 444.951} C_DIS
LIN {X 142.0336,Y 15.7588,Z 188,A 9.9254,B 2.066,C 0.1175,E1 2.2281,E2 443.7946} C_DIS
LIN {X 141.6057,Y 19.2338,Z 188,A 11.3442,B 2.0662,C 0.1134,E1 2.2276,E2 442.373} C_DIS
LIN {X 141.0925,Y 22.6985,Z 188,A 12.5795,B 2.0663,C 0.1109,E1 2.2271,E2 441.1597} C_DIS
LIN {X 140.491,Y 26.1607,Z 188,A 13.9005,B 2.0665,C 0.1077,E1 2.2264,E2 439.8498} C_DIS
LIN {X 139.8017,Y 29.6212,Z 188,A 15.216,B 2.0667,C 0.1046,E1 2.2257,E2 438.5469} C_DIS
LIN {X 139.0358,Y 33.0284,Z 188,A 16.616,B 2.0668,C 0.1007,E1 2.2248,E2 437.1462} C_DIS
LIN {X 138.1876,Y 36.4137,Z 188,A 17.838,B 2.067,C 0.0983,E1 2.224,E2 435.9471} C_DIS
LIN {X 137.2569,Y 39.7779,Z 188,A 19.1786,B 2.0671,C 0.095,E1 2.2229,E2 434.6137} C_DIS
LIN {X 136.2321,Y 43.157,Z 188,A 20.48,B 2.0673,C 0.0921,E1 2.2219,E2 433.327} C_DIS
LIN {X 135.1331,Y 46.4839,Z 188,A 21.8,B 2.0673,C 0.089,E1 2.2207,E2 432.0176} C_DIS
LIN {X 133.7739,Y 50.2606,Z 188,A 23.2148,B 2.0675,C 0.0862,E1 2.2194,E2 430.6279} C_DIS
LIN {X 132.6858,Y 53.0677,Z 188,A 24.5241,B 2.0677,C 0.0822,E1 2.218,E2 429.3045} C_DIS
LIN {X 131.346,Y 56.3025,Z 188,A 25.8138,B 2.0677,C 0.0794,E1 2.2166,E2 428.0295} C_DIS
LIN {X 129.9273,Y 59.5039,Z 188,A 27.0811,B 2.0679,C 0.0768,E1 2.2152,E2 426.7797} C_DIS
LIN {X 128.4305,Y 62.67,Z 188,A 28.4014,B 2.0679,C 0.0739,E1 2.2136,E2 425.4699} C_DIS
LIN {X 126.7502,Y 66.0013,Z 188,A 29.8601,B 2.0681,C 0.0704,E1 2.2117,E2 424.0157} C_DIS
LIN {X 124.7675,Y 69.6803,Z 188,A 31.5112,B 2.0682,C 0.0664,E1 2.2095,E2 422.3673} C_DIS
LIN {X 122.5736,Y 73.4708,Z 188,A 33.0876,B 2.0683,C 0.0634,E1 2.2073,E2 420.8139} C_DIS
LIN {X 120.2557,Y 77.2058,Z 188,A 34.7474,B 2.0684,C 0.0599,E1 2.2049,E2 419.167} C_DIS
LIN {X 117.8385,Y 80.8468,Z 188,A 36.4698,B 2.0685,C 0.0559,E1 2.2022,E2 417.448} C_DIS
LIN {X 115.1685,Y 84.607,Z 188,A 38.1452,B 2.0686,C 0.0529,E1 2.1995,E2 415.7948} C_DIS
LIN {X 112.6517,Y 87.9312,Z 188,A 39.8253,B 2.0687,C 0.049,E1 2.1966,E2 414.1134} C_DIS
LIN {X 109.7605,Y 91.5147,Z 188,A 41.5763,B 2.0687,C 0.0455,E1 2.1935,E2 412.3744} C_DIS
LIN {X 106.9066,Y 94.8322,Z 188,A 43.1881,B 2.0689,C 0.0427,E1 2.1906,E2 410.7807} C_DIS
LIN {X 103.9417,Y 98.0726,Z 188,A 44.8562,B 2.0689,C 0.0395,E1 2.1874,E2 409.1244} C_DIS
LIN {X 101.0499,Y 101.0507,Z 188,A 46.4247,B 2.0689,C 0.0367,E1 2.1844,E2 407.5681} C_DIS
LIN {X 97.9057,Y 104.0992,Z 188,A 48.0844,B 2.069,C 0.0338,E1 2.181,E2 405.9206} C_DIS
LIN {X 94.6594,Y 107.0594,Z 188,A 49.786,B 2.069,C 0.0307,E1 2.1775,E2 404.2265} C_DIS
LIN {X 91.3378,Y 109.9072,Z 188,A 51.449,B 2.0691,C 0.028,E1 2.174,E2 402.5751} C_DIS
LIN {X 87.9298,Y 112.6529,Z 188,A 53.2098,B 2.0691,C 0.0247,E1 2.1701,E2 400.8135} C_DIS
LIN {X 84.2285,Y 115.4465,Z 188,A 54.9886,B 2.0691,C 0.0219,E1 2.1662,E2 399.0451} C_DIS
LIN {X 80.6563,Y 117.9693,Z 188,A 56.6167,B 2.0692,C 0.0197,E1 2.1624,E2 397.4329} C_DIS
Enddeposition()
END
